  MoveL 6990 to (509.6, 509.6, 14.4) mm, rotated rx 0 ry 90 rz 0 deg; joints [-12.688, -27.581, 110.091, -16.755, -81.963, 51.382]
  Call Extruder(0.559)
  MoveL 6991 to (490.4, 509.6, 14.4) mm, rotated rx 0 ry 90 rz 0 deg; joints [-13.088, -27.943, 112.38, -17.087, -83.818, 50.861]
  MoveL 6992 to (490.4, 490.4, 14.4) mm, rotated rx 0 ry 90 rz 0 deg; joints [-11.303, -28.014, 112.87, -15.281, -84.175, 50.582]
  Call Extruder(0.146)
  MoveL 6993 to (495.43, 490.4, 14.4) mm, rotated rx 0 ry 90 rz 0 deg; joints [-11.21, -27.928, 112.274, -15.202, -83.681, 50.708]
  Call Extruder(0.010)
  MoveL 6994 to (495.78, 490.4, 14.4) mm, rotated rx 0 ry 90 rz 0 deg; joints [-11.203, -27.922, 112.232, -15.196, -83.646, 50.717]
  Call Extruder(0.007)
  MoveL 6995 to (495.78, 490.75, 14.4) mm, rotated rx 0 ry 90 rz 0 deg; joints [-11.236, -27.92, 112.224, -15.229, -83.64, 50.722]
  Call Extruder(0.035)
  MoveL 6996 to (495.78, 491.95, 14.4) mm, rotated rx 0 ry 90 rz 0 deg; joints [-11.347, -27.916, 112.196, -15.342, -83.62, 50.739]
  Call Extruder(0.010)
  MoveL 6997 to (495.78, 492.3, 14.4) mm, rotated rx 0 ry 90 rz 0 deg; joints [-11.38, -27.915, 112.187, -15.375, -83.614, 50.744]
  Call Extruder(0.007)
  MoveL 6998 to (496.13, 492.3, 14.4) mm, rotated rx 0 ry 90 rz 0 deg; joints [-11.373, -27.909, 112.146, -15.369, -83.58, 50.753]
  Call Extruder(0.061)
  MoveL 6999 to (498.23, 492.3, 14.4) mm, rotated rx 0 ry 90 rz 0 deg; joints [-11.334, -27.871, 111.895, -15.336, -83.373, 50.806]
  Call Extruder(0.055)
  MoveL 7000 to (498.23, 490.4, 14.4) mm, rotated rx 0 ry 90 rz 0 deg; joints [-11.158, -27.878, 111.94, -15.158, -83.405, 50.778]
  Call Extruder(0.082)
  MoveL 7001 to (501.04, 490.4, 14.4) mm, rotated rx 0 ry 90 rz 0 deg; joints [-11.107, -27.827, 111.605, -15.116, -83.13, 50.848]
  Call Extruder(0.055)
  MoveL 7002 to (501.04, 492.3, 14.4) mm, rotated rx 0 ry 90 rz 0 deg; joints [-11.282, -27.82, 111.56, -15.293, -83.098, 50.876]
  Call Extruder(0.061)
  MoveL 7003 to (503.12, 492.3, 14.4) mm, rotated rx 0 ry 90 rz 0 deg; joints [-11.244, -27.781, 111.31, -15.262, -82.893, 50.928]
  Call Extruder(0.007)
  MoveL 7004 to (503.48, 492.3, 14.4) mm, rotated rx 0 ry 90 rz 0 deg; joints [-11.238, -27.774, 111.268, -15.256, -82.859, 50.937]
  Set speed (120.0 mm/s)
  MoveL 7005 to (503.48, 491.95, 14.4) mm, rotated rx 0 ry 90 rz 0 deg; joints [-11.206, -27.775, 111.276, -15.224, -82.865, 50.931]
  Set speed (1000.0 mm/s)
  MoveL 7006 to (503.47, 491.9, 14.4) mm, rotated rx 0 ry 90 rz 0 deg; joints [-11.201, -27.775, 111.278, -15.219, -82.866, 50.931]
  Set speed (1000.0 mm/s)
  MoveL 7007 to (504.18, 491.9, 14.4) mm, rotated rx 0 ry 90 rz 0 deg; joints [-11.189, -27.762, 111.194, -15.209, -82.797, 50.948]
  Set speed (1000.0 mm/s)
  MoveL 7008 to (495.75, 492.33, 14.4) mm, rotated rx 0 ry 90 rz 0 deg; joints [-11.383, -27.915, 112.19, -15.378, -83.616, 50.744]
  Set speed (1000.0 mm/s)
  MoveL 7009 to (490.68, 490.68, 14.4) mm, rotated rx 0 ry 90 rz 0 deg; joints [-11.324, -28.008, 112.831, -15.303, -84.143, 50.593]
  Set speed (1000.0 mm/s)
  MoveL 7010 to (490.68, 490.68, 14.5) mm, rotated rx 0 ry 90 rz 0 deg; joints [-11.324, -28.019, 112.836, -15.303, -84.138, 50.594]
  Set speed (30.0 mm/s)
  Call Extruder(0.767)
  MoveL 7011 to (509.32, 509.32, 14.5) mm, rotated rx 0 ry 90 rz 0 deg; joints [-12.669, -27.598, 110.138, -16.734, -81.99, 51.371]
  MoveL 7012 to (509.44, 509.44, 14.5) mm, rotated rx 0 ry 90 rz 0 deg; joints [-12.677, -27.595, 110.12, -16.743, -81.976, 51.376]
  Set speed (120.0 mm/s)
  MoveL 7013 to (507.64, 503.83, 14.5) mm, rotated rx 0 ry 90 rz 0 deg; joints [-12.208, -27.657, 110.485, -16.258, -82.25, 51.231]
  Set speed (1000.0 mm/s)
  MoveL 7014 to (507.39, 502.51, 14.5) mm, rotated rx 0 ry 90 rz 0 deg; joints [-12.093, -27.667, 110.55, -16.14, -82.298, 51.202]
  Set speed (30.0 mm/s)
  Call Extruder(0.280)
  MoveL 7015 to (500.58, 509.32, 14.5) mm, rotated rx 0 ry 90 rz 0 deg; joints [-12.847, -27.771, 111.185, -16.88, -82.834, 51.137]
  Set speed (120.0 mm/s)
  MoveL 7016 to (499.42, 509.32, 14.5) mm, rotated rx 0 ry 90 rz 0 deg; joints [-12.872, -27.792, 111.324, -16.9, -82.946, 51.105]
  Set speed (30.0 mm/s)
  Call Extruder(0.360)
  MoveL 7017 to (490.68, 500.58, 14.5) mm, rotated rx 0 ry 90 rz 0 deg; joints [-12.247, -27.984, 112.592, -16.236, -83.959, 50.734]
  Set speed (120.0 mm/s)
  MoveL 7018 to (490.68, 499.42, 14.5) mm, rotated rx 0 ry 90 rz 0 deg; joints [-12.139, -27.988, 112.621, -16.127, -83.981, 50.717]
  Set speed (30.0 mm/s)
  Call Extruder(0.281)
  MoveL 7019 to (497.52, 492.58, 14.5) mm, rotated rx 0 ry 90 rz 0 deg; joints [-11.373, -27.894, 111.979, -15.374, -83.433, 50.794]
  Set speed (120.0 mm/s)
  MoveL 7020 to (498.45, 491.65, 14.5) mm, rotated rx 0 ry 90 rz 0 deg; joints [-11.269, -27.88, 111.889, -15.272, -83.357, 50.803]
  Set speed (30.0 mm/s)
  Call Extruder(0.040)
  MoveL 7021 to (499.42, 490.68, 14.5) mm, rotated rx 0 ry 90 rz 0 deg; joints [-11.163, -27.866, 111.797, -15.167, -83.279, 50.813]
  Set speed (120.0 mm/s)
  MoveL 7022 to (500.58, 490.68, 14.5) mm, rotated rx 0 ry 90 rz 0 deg; joints [-11.142, -27.845, 111.658, -15.149, -83.165, 50.842]
  Set speed (30.0 mm/s)
  Call Extruder(0.010)
  MoveL 7023 to (500.82, 490.92, 14.5) mm, rotated rx 0 ry 90 rz 0 deg; joints [-11.159, -27.839, 111.624, -15.168, -83.137, 50.852]
  Set speed (120.0 mm/s)
  MoveL 7024 to (501.08, 492.33, 14.5) mm, rotated rx 0 ry 90 rz 0 deg; joints [-11.284, -27.829, 111.56, -15.295, -83.089, 50.879]
  Set speed (1000.0 mm/s)
  MoveL 7025 to (502.48, 492.58, 14.5) mm, rotated rx 0 ry 90 rz 0 deg; joints [-11.282, -27.802, 111.386, -15.297, -82.947, 50.918]
  Set speed (30.0 mm/s)
  Call Extruder(0.202)
  MoveL 7026 to (507.39, 497.49, 14.5) mm, rotated rx 0 ry 90 rz 0 deg; joints [-11.639, -27.688, 110.677, -15.678, -82.384, 51.119]
  Set speed (120.0 mm/s)
  MoveL 7027 to (507.94, 498.04, 14.5) mm, rotated rx 0 ry 90 rz 0 deg; joints [-11.678, -27.675, 110.597, -15.72, -82.322, 51.141]
  Set speed (30.0 mm/s)
  Call Extruder(0.057)
  MoveL 7028 to (509.32, 499.42, 14.5) mm, rotated rx 0 ry 90 rz 0 deg; joints [-11.777, -27.642, 110.396, -15.826, -82.164, 51.199]
  Set speed (120.0 mm/s)
  MoveL 7029 to (509.32, 500.58, 14.5) mm, rotated rx 0 ry 90 rz 0 deg; joints [-11.882, -27.637, 110.367, -15.932, -82.144, 51.219]
  Set speed (30.0 mm/s)
  Call Extruder(0.018)
  MoveL 7030 to (508.87, 501.02, 14.5) mm, rotated rx 0 ry 90 rz 0 deg; joints [-11.931, -27.644, 110.409, -15.98, -82.18, 51.215]
  Set speed (120.0 mm/s)
  MoveL 7031 to (507.64, 497.79, 14.5) mm, rotated rx 0 ry 90 rz 0 deg; joints [-11.661, -27.682, 110.639, -15.701, -82.355, 51.13]
  Set speed (1000.0 mm/s)
  MoveL 7032 to (507.64, 495.21, 14.5) mm, rotated rx 0 ry 90 rz 0 deg; joints [-11.427, -27.692, 110.702, -15.464, -82.398, 51.088]
  Set speed (1000.0 mm/s)
  MoveL 7033 to (509.32, 490.68, 14.5) mm, rotated rx 0 ry 90 rz 0 deg; joints [-10.985, -27.677, 110.608, -15.021, -82.308, 51.056]
  Set speed (30.0 mm/s)
  Call Extruder(0.767)
  MoveL 7034 to (490.68, 509.32, 14.5) mm, rotated rx 0 ry 90 rz 0 deg; joints [-13.056, -27.95, 112.36, -17.056, -83.792, 50.865]
  MoveL 7035 to (490.56, 509.44, 14.5) mm, rotated rx 0 ry 90 rz 0 deg; joints [-13.07, -27.952, 112.371, -17.07, -83.801, 50.864]
  Set speed (120.0 mm/s)
  MoveL 7036 to (503.61, 492.37, 14.5) mm, rotated rx 0 ry 90 rz 0 deg; joints [-11.242, -27.782, 111.255, -15.261, -82.84, 50.943]
  Set speed (1000.0 mm/s)
  MoveL 7037 to (503.54, 492.3, 14.5) mm, rotated rx 0 ry 90 rz 0 deg; joints [-11.237, -27.783, 111.266, -15.255, -82.848, 50.94]
  Set speed (15.0 mm/s)
  Call Extruder(0.010)
  MoveL 7038 to (503.54, 491.95, 14.5) mm, rotated rx 0 ry 90 rz 0 deg; joints [-11.205, -27.785, 111.274, -15.223, -82.853, 50.934]
  Call Extruder(0.035)
  MoveL 7039 to (503.54, 490.75, 14.5) mm, rotated rx 0 ry 90 rz 0 deg; joints [-11.095, -27.789, 111.302, -15.111, -82.873, 50.916]
  Call Extruder(0.010)
  MoveL 7040 to (503.54, 490.4, 14.5) mm, rotated rx 0 ry 90 rz 0 deg; joints [-11.062, -27.79, 111.311, -15.079, -82.879, 50.911]
  Call Extruder(0.007)
  MoveL 7041 to (503.89, 490.4, 14.5) mm, rotated rx 0 ry 90 rz 0 deg; joints [-11.056, -27.784, 111.269, -15.074, -82.845, 50.919]
  Call Extruder(0.166)
  MoveL 7042 to (509.6, 490.4, 14.5) mm, rotated rx 0 ry 90 rz 0 deg; joints [-10.955, -27.672, 110.581, -14.991, -82.285, 51.058]
  Call Extruder(0.141)
  MoveL 7043 to (509.6, 495.24, 14.5) mm, rotated rx 0 ry 90 rz 0 deg; joints [-11.394, -27.653, 110.466, -15.437, -82.207, 51.137]
  Call Extruder(0.056)
  MoveL 7044 to (507.67, 495.24, 14.5) mm, rotated rx 0 ry 90 rz 0 deg; joints [-11.429, -27.692, 110.698, -15.466, -82.395, 51.089]
  Call Extruder(0.073)
  MoveL 7045 to (507.67, 497.76, 14.5) mm, rotated rx 0 ry 90 rz 0 deg; joints [-11.658, -27.682, 110.636, -15.698, -82.352, 51.13]
  Call Extruder(0.056)
  MoveL 7046 to (509.6, 497.76, 14.5) mm, rotated rx 0 ry 90 rz 0 deg; joints [-11.622, -27.643, 110.404, -15.669, -82.165, 51.179]
  Call Extruder(0.093)
  MoveL 7047 to (509.6, 500.95, 14.5) mm, rotated rx 0 ry 90 rz 0 deg; joints [-11.91, -27.63, 110.324, -15.963, -82.11, 51.232]
  Call Extruder(0.010)
  MoveL 7048 to (509.6, 501.3, 14.5) mm, rotated rx 0 ry 90 rz 0 deg; joints [-11.942, -27.628, 110.315, -15.995, -82.104, 51.238]
  Call Extruder(0.007)
  MoveL 7049 to (509.25, 501.3, 14.5) mm, rotated rx 0 ry 90 rz 0 deg; joints [-11.949, -27.635, 110.357, -16, -82.138, 51.229]
  Call Extruder(0.036)
  MoveL 7050 to (508.02, 501.3, 14.5) mm, rotated rx 0 ry 90 rz 0 deg; joints [-11.972, -27.66, 110.505, -16.019, -82.258, 51.198]
  Call Extruder(0.010)
  MoveL 7051 to (507.67, 501.3, 14.5) mm, rotated rx 0 ry 90 rz 0 deg; joints [-11.979, -27.667, 110.547, -16.024, -82.292, 51.189]
  Call Extruder(0.007)
  MoveL 7052 to (507.67, 501.65, 14.5) mm, rotated rx 0 ry 90 rz 0 deg; joints [-12.01, -27.665, 110.538, -16.057, -82.286, 51.195]
  Call Extruder(0.063)
  MoveL 7053 to (507.67, 503.81, 14.5) mm, rotated rx 0 ry 90 rz 0 deg; joints [-12.205, -27.656, 110.483, -16.255, -82.248, 51.231]
  Call Extruder(0.056)
  MoveL 7054 to (509.6, 503.81, 14.5) mm, rotated rx 0 ry 90 rz 0 deg; joints [-12.168, -27.617, 110.25, -16.225, -82.061, 51.281]
  Call Extruder(0.169)
  MoveL 7055 to (509.6, 509.6, 14.5) mm, rotated rx 0 ry 90 rz 0 deg; joints [-12.688, -27.591, 110.096, -16.755, -81.957, 51.383]
  Call Extruder(0.559)
  MoveL 7056 to (490.4, 509.6, 14.5) mm, rotated rx 0 ry 90 rz 0 deg; joints [-13.088, -27.954, 112.385, -17.088, -83.813, 50.862]
  MoveL 7057 to (490.4, 490.4, 14.5) mm, rotated rx 0 ry 90 rz 0 deg; joints [-11.303, -28.024, 112.875, -15.281, -84.17, 50.583]
  Call Extruder(0.145)
  MoveL 7058 to (495.37, 490.4, 14.5) mm, rotated rx 0 ry 90 rz 0 deg; joints [-11.211, -27.939, 112.286, -15.203, -83.681, 50.708]
  Call Extruder(0.010)
  MoveL 7059 to (495.72, 490.4, 14.5) mm, rotated rx 0 ry 90 rz 0 deg; joints [-11.204, -27.933, 112.244, -15.197, -83.646, 50.717]
  Call Extruder(0.007)
  MoveL 7060 to (495.72, 490.75, 14.5) mm, rotated rx 0 ry 90 rz 0 deg; joints [-11.237, -27.932, 112.236, -15.23, -83.641, 50.722]
  Call Extruder(0.035)
  MoveL 7061 to (495.72, 491.95, 14.5) mm, rotated rx 0 ry 90 rz 0 deg; joints [-11.348, -27.928, 112.208, -15.343, -83.62, 50.739]
  Call Extruder(0.010)
  MoveL 7062 to (495.72, 492.3, 14.5) mm, rotated rx 0 ry 90 rz 0 deg; joints [-11.381, -27.927, 112.199, -15.376, -83.614, 50.744]
  Call Extruder(0.007)
  MoveL 7063 to (496.07, 492.3, 14.5) mm, rotated rx 0 ry 90 rz 0 deg; joints [-11.374, -27.92, 112.158, -15.37, -83.58, 50.753]
  Call Extruder(0.061)
  MoveL 7064 to (498.17, 492.3, 14.5) mm, rotated rx 0 ry 90 rz 0 deg; joints [-11.335, -27.883, 111.907, -15.337, -83.373, 50.806]
  Call Extruder(0.055)
  MoveL 7065 to (498.18, 490.4, 14.5) mm, rotated rx 0 ry 90 rz 0 deg; joints [-11.159, -27.889, 111.952, -15.159, -83.405, 50.778]
  Call Extruder(0.085)
  MoveL 7066 to (501.1, 490.4, 14.5) mm, rotated rx 0 ry 90 rz 0 deg; joints [-11.106, -27.836, 111.602, -15.115, -83.118, 50.851]
  Call Extruder(0.055)
  MoveL 7067 to (501.1, 492.3, 14.5) mm, rotated rx 0 ry 90 rz 0 deg; joints [-11.281, -27.829, 111.557, -15.292, -83.086, 50.879]
  Call Extruder(0.061)
  MoveL 7068 to (503.19, 492.3, 14.5) mm, rotated rx 0 ry 90 rz 0 deg; joints [-11.243, -27.79, 111.307, -15.261, -82.882, 50.931]
  Call Extruder(0.007)
  MoveL 7069 to (503.54, 492.3, 14.5) mm, rotated rx 0 ry 90 rz 0 deg; joints [-11.237, -27.783, 111.266, -15.255, -82.848, 50.94]
  Set speed (120.0 mm/s)
  MoveL 7070 to (503.54, 491.95, 14.5) mm, rotated rx 0 ry 90 rz 0 deg; joints [-11.205, -27.785, 111.274, -15.223, -82.853, 50.934]
  Set speed (1000.0 mm/s)
  MoveL 7071 to (503.54, 491.9, 14.5) mm, rotated rx 0 ry 90 rz 0 deg; joints [-11.2, -27.785, 111.275, -15.218, -82.854, 50.934]
  Set speed (1000.0 mm/s)
  MoveL 7072 to (504.24, 491.9, 14.5) mm, rotated rx 0 ry 90 rz 0 deg; joints [-11.187, -27.771, 111.191, -15.208, -82.786, 50.951]
  Set speed (1000.0 mm/s)
  MoveL 7073 to (495.69, 492.33, 14.5) mm, rotated rx 0 ry 90 rz 0 deg; joints [-11.384, -27.927, 112.202, -15.379, -83.616, 50.744]
  Set speed (1000.0 mm/s)
  MoveL 7074 to (490.68, 490.68, 14.5) mm, rotated rx 0 ry 90 rz 0 deg; joints [-11.324, -28.019, 112.836, -15.303, -84.138, 50.594]
  Set speed (1000.0 mm/s)
  MoveL 7075 to (490.68, 490.68, 14.6) mm, rotated rx 0 ry 90 rz 0 deg; joints [-11.324, -28.029, 112.841, -15.303, -84.132, 50.596]
  Set speed (30.0 mm/s)
  Call Extruder(0.767)
  MoveL 7076 to (509.32, 509.32, 14.6) mm, rotated rx 0 ry 90 rz 0 deg; joints [-12.669, -27.609, 110.143, -16.734, -81.985, 51.372]
  MoveL 7077 to (509.44, 509.44, 14.6) mm, rotated rx 0 ry 90 rz 0 deg; joints [-12.677, -27.605, 110.125, -16.743, -81.97, 51.378]
  Set speed (120.0 mm/s)
  MoveL 7078 to (507.64, 503.89, 14.6) mm, rotated rx 0 ry 90 rz 0 deg; joints [-12.213, -27.667, 110.489, -16.263, -82.244, 51.234]
  Set speed (1000.0 mm/s)
  MoveL 7079 to (507.39, 502.51, 14.6) mm, rotated rx 0 ry 90 rz 0 deg; joints [-12.093, -27.678, 110.555, -16.14, -82.293, 51.204]
  Set speed (30.0 mm/s)
  Call Extruder(0.280)
  MoveL 7080 to (500.58, 509.32, 14.6) mm, rotated rx 0 ry 90 rz 0 deg; joints [-12.847, -27.781, 111.191, -16.88, -82.829, 51.138]
  Set speed (120.0 mm/s)
  MoveL 7081 to (499.42, 509.32, 14.6) mm, rotated rx 0 ry 90 rz 0 deg; joints [-12.872, -27.803, 111.329, -16.901, -82.941, 51.107]
  Set speed (30.0 mm/s)
  Call Extruder(0.360)
  MoveL 7082 to (490.68, 500.58, 14.6) mm, rotated rx 0 ry 90 rz 0 deg; joints [-12.247, -27.995, 112.597, -16.237, -83.954, 50.735]
  Set speed (120.0 mm/s)
  MoveL 7083 to (490.68, 499.42, 14.6) mm, rotated rx 0 ry 90 rz 0 deg; joints [-12.139, -27.999, 112.626, -16.128, -83.975, 50.718]
  Set speed (30.0 mm/s)
  Call Extruder(0.281)
  MoveL 7084 to (497.52, 492.58, 14.6) mm, rotated rx 0 ry 90 rz 0 deg; joints [-11.373, -27.904, 111.984, -15.374, -83.428, 50.795]
  Set speed (120.0 mm/s)
  MoveL 7085 to (498.4, 491.7, 14.6) mm, rotated rx 0 ry 90 rz 0 deg; joints [-11.276, -27.891, 111.9, -15.278, -83.356, 50.804]
  Set speed (30.0 mm/s)
  Call Extruder(0.042)
  MoveL 7086 to (499.42, 490.68, 14.6) mm, rotated rx 0 ry 90 rz 0 deg; joints [-11.163, -27.877, 111.802, -15.167, -83.273, 50.815]
  Set speed (120.0 mm/s)
  MoveL 7087 to (500.58, 490.68, 14.6) mm, rotated rx 0 ry 90 rz 0 deg; joints [-11.141, -27.855, 111.663, -15.149, -83.159, 50.843]
  Set speed (30.0 mm/s)
  Call Extruder(0.013)
  MoveL 7088 to (500.89, 490.99, 14.6) mm, rotated rx 0 ry 90 rz 0 deg; joints [-11.164, -27.848, 111.62, -15.173, -83.124, 50.855]
  Set speed (120.0 mm/s)
  MoveL 7089 to (502.48, 492.58, 14.6) mm, rotated rx 0 ry 90 rz 0 deg; joints [-11.282, -27.813, 111.391, -15.298, -82.941, 50.919]
  Set speed (30.0 mm/s)
  Call Extruder(0.202)
  MoveL 7090 to (507.39, 497.49, 14.6) mm, rotated rx 0 ry 90 rz 0 deg; joints [-11.639, -27.699, 110.681, -15.678, -82.379, 51.12]
  Set speed (120.0 mm/s)
  MoveL 7091 to (507.88, 497.98, 14.6) mm, rotated rx 0 ry 90 rz 0 deg; joints [-11.674, -27.687, 110.611, -15.716, -82.323, 51.14]
  Set speed (30.0 mm/s)
  Call Extruder(0.059)
  MoveL 7092 to (509.32, 499.42, 14.6) mm, rotated rx 0 ry 90 rz 0 deg; joints [-11.777, -27.652, 110.401, -15.826, -82.159, 51.201]
  Set speed (120.0 mm/s)
  MoveL 7093 to (509.32, 500.58, 14.6) mm, rotated rx 0 ry 90 rz 0 deg; joints [-11.882, -27.647, 110.372, -15.933, -82.139, 51.22]
  Set speed (30.0 mm/s)
  Call Extruder(0.021)
  MoveL 7094 to (508.82, 501.08, 14.6) mm, rotated rx 0 ry 90 rz 0 deg; joints [-11.937, -27.655, 110.42, -15.986, -82.179, 51.216]
  Set speed (120.0 mm/s)
  MoveL 7095 to (507.65, 497.73, 14.6) mm, rotated rx 0 ry 90 rz 0 deg; joints [-11.656, -27.693, 110.645, -15.696, -82.35, 51.13]
  Set speed (1000.0 mm/s)
  MoveL 7096 to (507.64, 495.15, 14.6) mm, rotated rx 0 ry 90 rz 0 deg; joints [-11.422, -27.703, 110.709, -15.458, -82.394, 51.088]
  Set speed (1000.0 mm/s)
  MoveL 7097 to (509.32, 490.68, 14.6) mm, rotated rx 0 ry 90 rz 0 deg; joints [-10.985, -27.687, 110.614, -15.021, -82.303, 51.057]
  Set speed (30.0 mm/s)
  Call Extruder(0.767)
  MoveL 7098 to (490.68, 509.32, 14.6) mm, rotated rx 0 ry 90 rz 0 deg; joints [-13.056, -27.961, 112.365, -17.056, -83.786, 50.867]
  MoveL 7099 to (490.56, 509.44, 14.6) mm, rotated rx 0 ry 90 rz 0 deg; joints [-13.07, -27.962, 112.376, -17.07, -83.796, 50.866]
  Set speed (120.0 mm/s)
  MoveL 7100 to (503.67, 492.37, 14.6) mm, rotated rx 0 ry 90 rz 0 deg; joints [-11.241, -27.791, 111.253, -15.26, -82.828, 50.946]
  Set speed (1000.0 mm/s)
  MoveL 7101 to (503.6, 492.3, 14.6) mm, rotated rx 0 ry 90 rz 0 deg; joints [-11.236, -27.793, 111.263, -15.255, -82.836, 50.943]
  Set speed (15.0 mm/s)
  Call Extruder(0.010)
  MoveL 7102 to (503.6, 491.95, 14.6) mm, rotated rx 0 ry 90 rz 0 deg; joints [-11.203, -27.794, 111.271, -15.222, -82.842, 50.937]
  Call Extruder(0.035)
  MoveL 7103 to (503.6, 490.75, 14.6) mm, rotated rx 0 ry 90 rz 0 deg; joints [-11.093, -27.798, 111.3, -15.111, -82.862, 50.919]
  Call Extruder(0.010)
  MoveL 7104 to (503.6, 490.4, 14.6) mm, rotated rx 0 ry 90 rz 0 deg; joints [-11.061, -27.8, 111.308, -15.078, -82.868, 50.914]
  Call Extruder(0.007)
  MoveL 7105 to (503.95, 490.4, 14.6) mm, rotated rx 0 ry 90 rz 0 deg; joints [-11.055, -27.793, 111.266, -15.073, -82.833, 50.922]
  Call Extruder(0.164)
  MoveL 7106 to (509.6, 490.4, 14.6) mm, rotated rx 0 ry 90 rz 0 deg; joints [-10.955, -27.683, 110.586, -14.991, -82.28, 51.06]
  Call Extruder(0.139)
  MoveL 7107 to (509.6, 495.18, 14.6) mm, rotated rx 0 ry 90 rz 0 deg; joints [-11.388, -27.664, 110.472, -15.432, -82.203, 51.137]
  Call Extruder(0.056)
  MoveL 7108 to (507.67, 495.18, 14.6) mm, rotated rx 0 ry 90 rz 0 deg; joints [-11.424, -27.702, 110.705, -15.46, -82.391, 51.089]
  Call Extruder(0.073)
  MoveL 7109 to (507.67, 497.7, 14.6) mm, rotated rx 0 ry 90 rz 0 deg; joints [-11.652, -27.692, 110.642, -15.693, -82.348, 51.131]
  Call Extruder(0.046)
  MoveL 7110 to (509.25, 497.7, 14.6) mm, rotated rx 0 ry 90 rz 0 deg; joints [-11.623, -27.661, 110.453, -15.669, -82.195, 51.17]
  Call Extruder(0.010)
  MoveL 7111 to (509.6, 497.7, 14.6) mm, rotated rx 0 ry 90 rz 0 deg; joints [-11.616, -27.654, 110.41, -15.664, -82.161, 51.179]
  Call Extruder(0.007)
  MoveL 7112 to (509.6, 498.05, 14.6) mm, rotated rx 0 ry 90 rz 0 deg; joints [-11.648, -27.652, 110.402, -15.696, -82.155, 51.185]
  Call Extruder(0.086)
  MoveL 7113 to (509.6, 501.01, 14.6) mm, rotated rx 0 ry 90 rz 0 deg; joints [-11.915, -27.64, 110.327, -15.968, -82.104, 51.235]
  Call Extruder(0.010)
  MoveL 7114 to (509.6, 501.36, 14.6) mm, rotated rx 0 ry 90 rz 0 deg; joints [-11.947, -27.638, 110.318, -16, -82.098, 51.241]
  Call Extruder(0.007)
  MoveL 7115 to (509.25, 501.36, 14.6) mm, rotated rx 0 ry 90 rz 0 deg; joints [-11.954, -27.645, 110.361, -16.006, -82.132, 51.232]
  Call Extruder(0.036)
  MoveL 7116 to (508.02, 501.36, 14.6) mm, rotated rx 0 ry 90 rz 0 deg; joints [-11.977, -27.67, 110.509, -16.024, -82.252, 51.2]
  Call Extruder(0.010)
  MoveL 7117 to (507.67, 501.36, 14.6) mm, rotated rx 0 ry 90 rz 0 deg; joints [-11.984, -27.677, 110.551, -16.03, -82.286, 51.191]
  Call Extruder(0.007)
  MoveL 7118 to (507.67, 501.71, 14.6) mm, rotated rx 0 ry 90 rz 0 deg; joints [-12.015, -27.676, 110.542, -16.062, -82.28, 51.197]
  Call Extruder(0.063)
  MoveL 7119 to (507.67, 503.86, 14.6) mm, rotated rx 0 ry 90 rz 0 deg; joints [-12.21, -27.666, 110.486, -16.26, -82.242, 51.234]
  Call Extruder(0.056)
  MoveL 7120 to (509.6, 503.87, 14.6) mm, rotated rx 0 ry 90 rz 0 deg; joints [-12.173, -27.627, 110.254, -16.23, -82.055, 51.284]
  Call Extruder(0.167)
  MoveL 7121 to (509.6, 509.6, 14.6) mm, rotated rx 0 ry 90 rz 0 deg; joints [-12.688, -27.602, 110.101, -16.755, -81.952, 51.385]
  Call Extruder(0.559)
  MoveL 7122 to (490.4, 509.6, 14.6) mm, rotated rx 0 ry 90 rz 0 deg; joints [-13.088, -27.965, 112.39, -17.088, -83.808, 50.864]
  MoveL 7123 to (490.4, 490.4, 14.6) mm, rotated rx 0 ry 90 rz 0 deg; joints [-11.303, -28.035, 112.881, -15.281, -84.165, 50.585]
  Call Extruder(0.143)
  MoveL 7124 to (495.31, 490.4, 14.6) mm, rotated rx 0 ry 90 rz 0 deg; joints [-11.212, -27.951, 112.298, -15.204, -83.681, 50.708]
  Call Extruder(0.010)
  MoveL 7125 to (495.66, 490.4, 14.6) mm, rotated rx 0 ry 90 rz 0 deg; joints [-11.205, -27.945, 112.256, -15.198, -83.647, 50.717]
  Call Extruder(0.007)
  MoveL 7126 to (495.66, 490.75, 14.6) mm, rotated rx 0 ry 90 rz 0 deg; joints [-11.238, -27.944, 112.248, -15.231, -83.641, 50.722]
  Call Extruder(0.035)
  MoveL 7127 to (495.66, 491.95, 14.6) mm, rotated rx 0 ry 90 rz 0 deg; joints [-11.349, -27.939, 112.22, -15.344, -83.621, 50.739]
  Call Extruder(0.010)
  MoveL 7128 to (495.66, 492.3, 14.6) mm, rotated rx 0 ry 90 rz 0 deg; joints [-11.382, -27.938, 112.211, -15.377, -83.615, 50.744]
  Call Extruder(0.007)
  MoveL 7129 to (496.01, 492.3, 14.6) mm, rotated rx 0 ry 90 rz 0 deg; joints [-11.375, -27.932, 112.17, -15.371, -83.58, 50.753]
  Call Extruder(0.061)
  MoveL 7130 to (498.12, 492.3, 14.6) mm, rotated rx 0 ry 90 rz 0 deg; joints [-11.336, -27.894, 111.919, -15.339, -83.374, 50.806]
  Call Extruder(0.055)
  MoveL 7131 to (498.12, 490.4, 14.6) mm, rotated rx 0 ry 90 rz 0 deg; joints [-11.16, -27.901, 111.964, -15.16, -83.406, 50.778]
  Call Extruder(0.089)
  MoveL 7132 to (501.16, 490.4, 14.6) mm, rotated rx 0 ry 90 rz 0 deg; joints [-11.105, -27.845, 111.6, -15.114, -83.107, 50.854]
  Call Extruder(0.055)
  MoveL 7133 to (501.17, 492.3, 14.6) mm, rotated rx 0 ry 90 rz 0 deg; joints [-11.28, -27.838, 111.555, -15.292, -83.075, 50.882]
  Call Extruder(0.061)
  MoveL 7134 to (503.25, 492.3, 14.6) mm, rotated rx 0 ry 90 rz 0 deg; joints [-11.242, -27.799, 111.305, -15.26, -82.87, 50.934]
  Call Extruder(0.007)
  MoveL 7135 to (503.6, 492.3, 14.6) mm, rotated rx 0 ry 90 rz 0 deg; joints [-11.236, -27.793, 111.263, -15.255, -82.836, 50.943]
  Set speed (120.0 mm/s)
  MoveL 7136 to (503.6, 491.95, 14.6) mm, rotated rx 0 ry 90 rz 0 deg; joints [-11.203, -27.794, 111.271, -15.222, -82.842, 50.937]
  Set speed (1000.0 mm/s)
  MoveL 7137 to (503.6, 491.9, 14.6) mm, rotated rx 0 ry 90 rz 0 deg; joints [-11.199, -27.794, 111.272, -15.218, -82.843, 50.937]
  Set speed (1000.0 mm/s)
  MoveL 7138 to (504.3, 491.9, 14.6) mm, rotated rx 0 ry 90 rz 0 deg; joints [-11.186, -27.781, 111.188, -15.207, -82.774, 50.954]
  Set speed (1000.0 mm/s)
  MoveL 7139 to (495.63, 492.33, 14.6) mm, rotated rx 0 ry 90 rz 0 deg; joints [-11.385, -27.939, 112.214, -15.38, -83.617, 50.744]
  Set speed (1000.0 mm/s)
  MoveL 7140 to (490.68, 490.68, 14.6) mm, rotated rx 0 ry 90 rz 0 deg; joints [-11.324, -28.029, 112.841, -15.303, -84.132, 50.596]
  Set speed (1000.0 mm/s)
  MoveL 7141 to (490.68, 490.68, 14.7) mm, rotated rx 0 ry 90 rz 0 deg; joints [-11.324, -28.04, 112.846, -15.303, -84.127, 50.597]
  Set speed (30.0 mm/s)
  Call Extruder(0.767)
  MoveL 7142 to (509.32, 509.32, 14.7) mm, rotated rx 0 ry 90 rz 0 deg; joints [-12.669, -27.619, 110.148, -16.734, -81.979, 51.374]
  MoveL 7143 to (509.44, 509.44, 14.7) mm, rotated rx 0 ry 90 rz 0 deg; joints [-12.677, -27.616, 110.13, -16.743, -81.965, 51.379]
  Set speed (120.0 mm/s)
  MoveL 7144 to (507.64, 503.95, 14.7) mm, rotated rx 0 ry 90 rz 0 deg; joints [-12.218, -27.677, 110.493, -16.269, -82.238, 51.236]
  Set speed (1000.0 mm/s)
  MoveL 7145 to (507.39, 502.51, 14.7) mm, rotated rx 0 ry 90 rz 0 deg; joints [-12.093, -27.688, 110.56, -16.14, -82.288, 51.205]
  Set speed (30.0 mm/s)
  Call Extruder(0.280)
  MoveL 7146 to (500.58, 509.32, 14.7) mm, rotated rx 0 ry 90 rz 0 deg; joints [-12.847, -27.792, 111.196, -16.881, -82.823, 51.14]
  Set speed (120.0 mm/s)
  MoveL 7147 to (499.42, 509.32, 14.7) mm, rotated rx 0 ry 90 rz 0 deg; joints [-12.872, -27.814, 111.334, -16.901, -82.935, 51.108]
  Set speed (30.0 mm/s)
  Call Extruder(0.360)
  MoveL 7148 to (490.68, 500.58, 14.7) mm, rotated rx 0 ry 90 rz 0 deg; joints [-12.247, -28.005, 112.602, -16.237, -83.949, 50.737]
  Set speed (120.0 mm/s)
  MoveL 7149 to (490.68, 499.42, 14.7) mm, rotated rx 0 ry 90 rz 0 deg; joints [-12.139, -28.009, 112.631, -16.128, -83.97, 50.72]
  Set speed (30.0 mm/s)
  Call Extruder(0.281)
  MoveL 7150 to (497.52, 492.58, 14.7) mm, rotated rx 0 ry 90 rz 0 deg; joints [-11.373, -27.915, 111.989, -15.374, -83.423, 50.797]
  Set speed (120.0 mm/s)
  MoveL 7151 to (498.34, 491.76, 14.7) mm, rotated rx 0 ry 90 rz 0 deg; joints [-11.282, -27.903, 111.91, -15.284, -83.356, 50.805]
  Set speed (30.0 mm/s)
  Call Extruder(0.044)
  MoveL 7152 to (499.42, 490.68, 14.7) mm, rotated rx 0 ry 90 rz 0 deg; joints [-11.163, -27.887, 111.807, -15.167, -83.268, 50.816]
  Set speed (120.0 mm/s)
  MoveL 7153 to (500.58, 490.68, 14.7) mm, rotated rx 0 ry 90 rz 0 deg; joints [-11.142, -27.866, 111.669, -15.149, -83.154, 50.845]
  Set speed (30.0 mm/s)
  Call Extruder(0.015)
  MoveL 7154 to (500.95, 491.05, 14.7) mm, rotated rx 0 ry 90 rz 0 deg; joints [-11.169, -27.858, 111.616, -15.178, -83.112, 50.859]
  Set speed (120.0 mm/s)
  MoveL 7155 to (502.48, 492.58, 14.7) mm, rotated rx 0 ry 90 rz 0 deg; joints [-11.282, -27.823, 111.396, -15.298, -82.936, 50.921]
  Set speed (30.0 mm/s)
  Call Extruder(0.202)
  MoveL 7156 to (507.39, 497.49, 14.7) mm, rotated rx 0 ry 90 rz 0 deg; joints [-11.639, -27.709, 110.687, -15.678, -82.374, 51.122]
  Set speed (120.0 mm/s)
  MoveL 7157 to (507.82, 497.92, 14.7) mm, rotated rx 0 ry 90 rz 0 deg; joints [-11.67, -27.699, 110.624, -15.711, -82.325, 51.139]
  Set speed (30.0 mm/s)
  Call Extruder(0.062)
  MoveL 7158 to (509.32, 499.42, 14.7) mm, rotated rx 0 ry 90 rz 0 deg; joints [-11.777, -27.663, 110.406, -15.826, -82.154, 51.202]
  Set speed (120.0 mm/s)
  MoveL 7159 to (509.32, 500.58, 14.7) mm, rotated rx 0 ry 90 rz 0 deg; joints [-11.882, -27.658, 110.377, -15.933, -82.134, 51.222]
  Set speed (30.0 mm/s)
  Call Extruder(0.023)
  MoveL 7160 to (508.76, 501.13, 14.7) mm, rotated rx 0 ry 90 rz 0 deg; joints [-11.943, -27.667, 110.43, -15.993, -82.178, 51.217]
  Set speed (120.0 mm/s)
  MoveL 7161 to (507.65, 497.67, 14.7) mm, rotated rx 0 ry 90 rz 0 deg; joints [-11.65, -27.703, 110.652, -15.691, -82.346, 51.131]
  Set speed (1000.0 mm/s)
  MoveL 7162 to (507.64, 495.09, 14.7) mm, rotated rx 0 ry 90 rz 0 deg; joints [-11.416, -27.714, 110.715, -15.453, -82.39, 51.089]
  Set speed (1000.0 mm/s)
  MoveL 7163 to (509.32, 490.68, 14.7) mm, rotated rx 0 ry 90 rz 0 deg; joints [-10.985, -27.698, 110.619, -15.021, -82.298, 51.059]
  Set speed (30.0 mm/s)
  Call Extruder(0.767)
  MoveL 7164 to (490.68, 509.32, 14.7) mm, rotated rx 0 ry 90 rz 0 deg; joints [-13.056, -27.972, 112.37, -17.056, -83.781, 50.869]
  MoveL 7165 to (490.56, 509.44, 14.7) mm, rotated rx 0 ry 90 rz 0 deg; joints [-13.07, -27.973, 112.381, -17.07, -83.791, 50.867]
  Set speed (120.0 mm/s)
  MoveL 7166 to (503.74, 492.37, 14.7) mm, rotated rx 0 ry 90 rz 0 deg; joints [-11.239, -27.8, 111.25, -15.259, -82.817, 50.949]
  Set speed (1000.0 mm/s)
  MoveL 7167 to (503.67, 492.3, 14.7) mm, rotated rx 0 ry 90 rz 0 deg; joints [-11.234, -27.802, 111.26, -15.254, -82.825, 50.946]
  Set speed (15.0 mm/s)
  Call Extruder(0.010)
  MoveL 7168 to (503.67, 491.95, 14.7) mm, rotated rx 0 ry 90 rz 0 deg; joints [-11.202, -27.803, 111.269, -15.221, -82.83, 50.94]
  Call Extruder(0.035)
  MoveL 7169 to (503.67, 490.75, 14.7) mm, rotated rx 0 ry 90 rz 0 deg; joints [-11.092, -27.808, 111.297, -15.11, -82.85, 50.922]
  Call Extruder(0.010)
  MoveL 7170 to (503.66, 490.4, 14.7) mm, rotated rx 0 ry 90 rz 0 deg; joints [-11.06, -27.809, 111.306, -15.077, -82.856, 50.917]
  Call Extruder(0.007)
  MoveL 7171 to (504.02, 490.4, 14.7) mm, rotated rx 0 ry 90 rz 0 deg; joints [-11.054, -27.802, 111.264, -15.072, -82.822, 50.925]
  Call Extruder(0.163)
  MoveL 7172 to (509.6, 490.4, 14.7) mm, rotated rx 0 ry 90 rz 0 deg; joints [-10.955, -27.693, 110.591, -14.991, -82.275, 51.061]
  Call Extruder(0.137)
  MoveL 7173 to (509.6, 495.12, 14.7) mm, rotated rx 0 ry 90 rz 0 deg; joints [-11.383, -27.675, 110.479, -15.426, -82.198, 51.138]
  Call Extruder(0.056)
  MoveL 7174 to (507.67, 495.12, 14.7) mm, rotated rx 0 ry 90 rz 0 deg; joints [-11.418, -27.713, 110.711, -15.455, -82.386, 51.09]
  Call Extruder(0.073)
  MoveL 7175 to (507.67, 497.64, 14.7) mm, rotated rx 0 ry 90 rz 0 deg; joints [-11.647, -27.703, 110.649, -15.688, -82.344, 51.131]
  Call Extruder(0.056)
  MoveL 7176 to (509.6, 497.64, 14.7) mm, rotated rx 0 ry 90 rz 0 deg; joints [-11.611, -27.664, 110.417, -15.659, -82.156, 51.18]
  Call Extruder(0.100)
  MoveL 7177 to (509.6, 501.07, 14.7) mm, rotated rx 0 ry 90 rz 0 deg; joints [-11.921, -27.65, 110.331, -15.973, -82.098, 51.237]
  Call Extruder(0.010)
  MoveL 7178 to (509.6, 501.42, 14.7) mm, rotated rx 0 ry 90 rz 0 deg; joints [-11.952, -27.648, 110.322, -16.006, -82.092, 51.243]
  Call Extruder(0.007)
  MoveL 7179 to (509.25, 501.42, 14.7) mm, rotated rx 0 ry 90 rz 0 deg; joints [-11.959, -27.656, 110.364, -16.011, -82.126, 51.234]
  Call Extruder(0.036)
  MoveL 7180 to (508.02, 501.41, 14.7) mm, rotated rx 0 ry 90 rz 0 deg; joints [-11.982, -27.68, 110.512, -16.03, -82.246, 51.203]
  Call Extruder(0.010)
  MoveL 7181 to (507.67, 501.41, 14.7) mm, rotated rx 0 ry 90 rz 0 deg; joints [-11.989, -27.687, 110.555, -16.035, -82.28, 51.194]
  Call Extruder(0.007)
  MoveL 7182 to (507.67, 501.76, 14.7) mm, rotated rx 0 ry 90 rz 0 deg; joints [-12.02, -27.686, 110.546, -16.067, -82.273, 51.2]
  Call Extruder(0.063)
  MoveL 7183 to (507.67, 503.92, 14.7) mm, rotated rx 0 ry 90 rz 0 deg; joints [-12.215, -27.677, 110.49, -16.266, -82.236, 51.236]
  Call Extruder(0.056)
  MoveL 7184 to (509.6, 503.92, 14.7) mm, rotated rx 0 ry 90 rz 0 deg; joints [-12.178, -27.638, 110.258, -16.235, -82.049, 51.286]
  Call Extruder(0.000)
  MoveL 7185 to (509.6, 503.92, 14.7) mm, rotated rx 0 ry 90 rz 0 deg; joints [-12.178, -27.638, 110.257, -16.235, -82.049, 51.286]
  Call Extruder(0.165)
  MoveL 7186 to (509.6, 509.6, 14.7) mm, rotated rx 0 ry 90 rz 0 deg; joints [-12.688, -27.612, 110.107, -16.755, -81.947, 51.386]
  Call Extruder(0.559)
  MoveL 7187 to (490.4, 509.6, 14.7) mm, rotated rx 0 ry 90 rz 0 deg; joints [-13.088, -27.975, 112.395, -17.088, -83.803, 50.865]
  MoveL 7188 to (490.4, 490.4, 14.7) mm, rotated rx 0 ry 90 rz 0 deg; joints [-11.303, -28.046, 112.886, -15.282, -84.159, 50.586]
  Call Extruder(0.141)
  MoveL 7189 to (495.26, 490.4, 14.7) mm, rotated rx 0 ry 90 rz 0 deg; joints [-11.213, -27.963, 112.31, -15.205, -83.681, 50.709]
  Call Extruder(0.010)
  MoveL 7190 to (495.61, 490.4, 14.7) mm, rotated rx 0 ry 90 rz 0 deg; joints [-11.206, -27.956, 112.268, -15.199, -83.647, 50.717]
  Call Extruder(0.007)
  MoveL 7191 to (495.61, 490.75, 14.7) mm, rotated rx 0 ry 90 rz 0 deg; joints [-11.239, -27.955, 112.26, -15.232, -83.641, 50.722]
  Call Extruder(0.035)
  MoveL 7192 to (495.61, 491.95, 14.7) mm, rotated rx 0 ry 90 rz 0 deg; joints [-11.35, -27.951, 112.231, -15.345, -83.621, 50.739]
  Call Extruder(0.010)
  MoveL 7193 to (495.61, 492.3, 14.7) mm, rotated rx 0 ry 90 rz 0 deg; joints [-11.383, -27.95, 112.223, -15.378, -83.615, 50.744]
  Call Extruder(0.007)
  MoveL 7194 to (495.96, 492.3, 14.7) mm, rotated rx 0 ry 90 rz 0 deg; joints [-11.376, -27.944, 112.181, -15.372, -83.58, 50.753]
  Call Extruder(0.061)
  MoveL 7195 to (498.06, 492.3, 14.7) mm, rotated rx 0 ry 90 rz 0 deg; joints [-11.337, -27.906, 111.931, -15.34, -83.374, 50.806]
  Call Extruder(0.055)
  MoveL 7196 to (498.06, 490.4, 14.7) mm, rotated rx 0 ry 90 rz 0 deg; joints [-11.162, -27.913, 111.976, -15.161, -83.406, 50.778]
  Call Extruder(0.092)
  MoveL 7197 to (501.23, 490.4, 14.7) mm, rotated rx 0 ry 90 rz 0 deg; joints [-11.104, -27.855, 111.598, -15.114, -83.095, 50.857]
  Call Extruder(0.055)
  MoveL 7198 to (501.23, 492.3, 14.7) mm, rotated rx 0 ry 90 rz 0 deg; joints [-11.279, -27.848, 111.552, -15.291, -83.063, 50.885]
  Call Extruder(0.061)
  MoveL 7199 to (503.32, 492.3, 14.7) mm, rotated rx 0 ry 90 rz 0 deg; joints [-11.241, -27.809, 111.302, -15.259, -82.859, 50.937]
  Call Extruder(0.007)
  MoveL 7200 to (503.67, 492.3, 14.7) mm, rotated rx 0 ry 90 rz 0 deg; joints [-11.234, -27.802, 111.26, -15.254, -82.825, 50.946]
  Set speed (120.0 mm/s)
  MoveL 7201 to (503.67, 491.95, 14.7) mm, rotated rx 0 ry 90 rz 0 deg; joints [-11.202, -27.803, 111.269, -15.221, -82.83, 50.94]
  Set speed (1000.0 mm/s)
  MoveL 7202 to (503.67, 491.9, 14.7) mm, rotated rx 0 ry 90 rz 0 deg; joints [-11.198, -27.803, 111.27, -15.217, -82.831, 50.94]
  Set speed (1000.0 mm/s)
  MoveL 7203 to (504.37, 491.9, 14.7) mm, rotated rx 0 ry 90 rz 0 deg; joints [-11.185, -27.79, 111.186, -15.206, -82.763, 50.957]
  Set speed (1000.0 mm/s)
  MoveL 7204 to (495.58, 492.33, 14.7) mm, rotated rx 0 ry 90 rz 0 deg; joints [-11.386, -27.95, 112.226, -15.381, -83.617, 50.744]
  Set speed (1000.0 mm/s)
  MoveL 7205 to (490.68, 490.68, 14.7) mm, rotated rx 0 ry 90 rz 0 deg; joints [-11.324, -28.04, 112.846, -15.303, -84.127, 50.597]
  Set speed (1000.0 mm/s)
  MoveL 7206 to (490.68, 490.68, 14.8) mm, rotated rx 0 ry 90 rz 0 deg; joints [-11.324, -28.051, 112.851, -15.304, -84.122, 50.599]
  Set speed (30.0 mm/s)
  Call Extruder(0.767)
  MoveL 7207 to (509.32, 509.32, 14.8) mm, rotated rx 0 ry 90 rz 0 deg; joints [-12.669, -27.629, 110.153, -16.734, -81.974, 51.375]
  MoveL 7208 to (509.44, 509.44, 14.8) mm, rotated rx 0 ry 90 rz 0 deg; joints [-12.677, -27.626, 110.135, -16.744, -81.96, 51.381]
  Set speed (120.0 mm/s)
  MoveL 7209 to (507.64, 504, 14.8) mm, rotated rx 0 ry 90 rz 0 deg; joints [-12.223, -27.687, 110.496, -16.274, -82.232, 51.238]
  Set speed (1000.0 mm/s)
  MoveL 7210 to (507.39, 502.51, 14.8) mm, rotated rx 0 ry 90 rz 0 deg; joints [-12.093, -27.699, 110.565, -16.141, -82.283, 51.207]
  Set speed (30.0 mm/s)
  Call Extruder(0.280)
  MoveL 7211 to (500.58, 509.32, 14.8) mm, rotated rx 0 ry 90 rz 0 deg; joints [-12.847, -27.802, 111.201, -16.881, -82.818, 51.141]
  Set speed (120.0 mm/s)
  MoveL 7212 to (499.42, 509.32, 14.8) mm, rotated rx 0 ry 90 rz 0 deg; joints [-12.872, -27.824, 111.339, -16.901, -82.93, 51.11]
  Set speed (30.0 mm/s)
  Call Extruder(0.360)
  MoveL 7213 to (490.68, 500.58, 14.8) mm, rotated rx 0 ry 90 rz 0 deg; joints [-12.247, -28.016, 112.607, -16.237, -83.943, 50.738]
  Set speed (120.0 mm/s)
  MoveL 7214 to (490.68, 499.42, 14.8) mm, rotated rx 0 ry 90 rz 0 deg; joints [-12.139, -28.02, 112.637, -16.128, -83.965, 50.722]
  Set speed (30.0 mm/s)
  Call Extruder(0.281)
  MoveL 7215 to (497.52, 492.58, 14.8) mm, rotated rx 0 ry 90 rz 0 deg; joints [-11.373, -27.925, 111.994, -15.374, -83.417, 50.798]
  Set speed (120.0 mm/s)
  MoveL 7216 to (498.28, 491.81, 14.8) mm, rotated rx 0 ry 90 rz 0 deg; joints [-11.288, -27.914, 111.921, -15.291, -83.355, 50.806]
  Set speed (30.0 mm/s)
  Call Extruder(0.047)
  MoveL 7217 to (499.42, 490.68, 14.8) mm, rotated rx 0 ry 90 rz 0 deg; joints [-11.163, -27.898, 111.812, -15.167, -83.263, 50.818]
  Set speed (120.0 mm/s)
  MoveL 7218 to (500.58, 490.68, 14.8) mm, rotated rx 0 ry 90 rz 0 deg; joints [-11.141, -27.876, 111.674, -15.149, -83.149, 50.846]
  Set speed (30.0 mm/s)
  Call Extruder(0.018)
  MoveL 7219 to (501.01, 491.11, 14.8) mm, rotated rx 0 ry 90 rz 0 deg; joints [-11.173, -27.867, 111.612, -15.183, -83.099, 50.863]
  Set speed (120.0 mm/s)
  MoveL 7220 to (502.48, 492.58, 14.8) mm, rotated rx 0 ry 90 rz 0 deg; joints [-11.282, -27.834, 111.401, -15.298, -82.931, 50.922]
  Set speed (30.0 mm/s)
  Call Extruder(0.202)
  MoveL 7221 to (507.39, 497.49, 14.8) mm, rotated rx 0 ry 90 rz 0 deg; joints [-11.639, -27.72, 110.692, -15.678, -82.369, 51.123]
  Set speed (120.0 mm/s)
  MoveL 7222 to (507.76, 497.86, 14.8) mm, rotated rx 0 ry 90 rz 0 deg; joints [-11.666, -27.711, 110.638, -15.707, -82.326, 51.138]
  Set speed (30.0 mm/s)
  Call Extruder(0.064)
  MoveL 7223 to (509.32, 499.42, 14.8) mm, rotated rx 0 ry 90 rz 0 deg; joints [-11.777, -27.673, 110.412, -15.827, -82.148, 51.204]
  Set speed (120.0 mm/s)
  MoveL 7224 to (509.32, 500.58, 14.8) mm, rotated rx 0 ry 90 rz 0 deg; joints [-11.882, -27.668, 110.382, -15.933, -82.129, 51.223]
  Set speed (30.0 mm/s)
  Call Extruder(0.025)
  MoveL 7225 to (508.71, 501.19, 14.8) mm, rotated rx 0 ry 90 rz 0 deg; joints [-11.949, -27.678, 110.44, -15.999, -82.177, 51.218]
  Set speed (120.0 mm/s)
  MoveL 7226 to (507.65, 497.61, 14.8) mm, rotated rx 0 ry 90 rz 0 deg; joints [-11.645, -27.714, 110.658, -15.686, -82.342, 51.131]
  Set speed (1000.0 mm/s)
  MoveL 7227 to (507.65, 495.03, 14.8) mm, rotated rx 0 ry 90 rz 0 deg; joints [-11.411, -27.725, 110.722, -15.447, -82.385, 51.089]
  Set speed (1000.0 mm/s)
  MoveL 7228 to (509.32, 490.68, 14.8) mm, rotated rx 0 ry 90 rz 0 deg; joints [-10.985, -27.708, 110.624, -15.021, -82.293, 51.06]
  Set speed (30.0 mm/s)
  Call Extruder(0.767)
  MoveL 7229 to (490.68, 509.32, 14.8) mm, rotated rx 0 ry 90 rz 0 deg; joints [-13.056, -27.982, 112.375, -17.057, -83.776, 50.87]
  MoveL 7230 to (490.56, 509.44, 14.8) mm, rotated rx 0 ry 90 rz 0 deg; joints [-13.07, -27.984, 112.386, -17.07, -83.785, 50.869]
  Set speed (120.0 mm/s)
  MoveL 7231 to (507.6, 501.4, 14.8) mm, rotated rx 0 ry 90 rz 0 deg; joints [-11.989, -27.699, 110.568, -16.035, -82.281, 51.193]
  Set speed (1000.0 mm/s)
  MoveL 7232 to (507.67, 501.47, 14.8) mm, rotated rx 0 ry 90 rz 0 deg; joints [-11.994, -27.698, 110.558, -16.04, -82.273, 51.196]
  Set speed (15.0 mm/s)
  Call Extruder(0.010)
  MoveL 7233 to (507.67, 501.82, 14.8) mm, rotated rx 0 ry 90 rz 0 deg; joints [-12.025, -27.696, 110.549, -16.073, -82.267, 51.202]
  Call Extruder(0.063)
  MoveL 7234 to (507.67, 503.98, 14.8) mm, rotated rx 0 ry 90 rz 0 deg; joints [-12.22, -27.687, 110.494, -16.271, -82.23, 51.239]
  Call Extruder(0.056)
  MoveL 7235 to (509.6, 503.98, 14.8) mm, rotated rx 0 ry 90 rz 0 deg; joints [-12.183, -27.648, 110.261, -16.241, -82.042, 51.289]
  Call Extruder(0.164)
  MoveL 7236 to (509.6, 509.6, 14.8) mm, rotated rx 0 ry 90 rz 0 deg; joints [-12.688, -27.622, 110.112, -16.756, -81.942, 51.388]
  Call Extruder(0.559)
  MoveL 7237 to (490.4, 509.6, 14.8) mm, rotated rx 0 ry 90 rz 0 deg; joints [-13.088, -27.986, 112.401, -17.088, -83.797, 50.867]
  MoveL 7238 to (490.4, 490.4, 14.8) mm, rotated rx 0 ry 90 rz 0 deg; joints [-11.303, -28.056, 112.891, -15.282, -84.154, 50.588]
  Call Extruder(0.140)
  MoveL 7239 to (495.2, 490.4, 14.8) mm, rotated rx 0 ry 90 rz 0 deg; joints [-11.214, -27.974, 112.321, -15.206, -83.682, 50.709]
  Call Extruder(0.010)
  MoveL 7240 to (495.55, 490.4, 14.8) mm, rotated rx 0 ry 90 rz 0 deg; joints [-11.208, -27.968, 112.28, -15.2, -83.647, 50.717]
  Call Extruder(0.007)
  MoveL 7241 to (495.55, 490.75, 14.8) mm, rotated rx 0 ry 90 rz 0 deg; joints [-11.24, -27.967, 112.272, -15.233, -83.641, 50.722]
  Call Extruder(0.035)
  MoveL 7242 to (495.55, 491.95, 14.8) mm, rotated rx 0 ry 90 rz 0 deg; joints [-11.352, -27.963, 112.243, -15.346, -83.621, 50.739]
  Call Extruder(0.010)
  MoveL 7243 to (495.55, 492.3, 14.8) mm, rotated rx 0 ry 90 rz 0 deg; joints [-11.384, -27.961, 112.235, -15.379, -83.615, 50.745]
  Call Extruder(0.007)
  MoveL 7244 to (495.9, 492.3, 14.8) mm, rotated rx 0 ry 90 rz 0 deg; joints [-11.377, -27.955, 112.193, -15.373, -83.581, 50.753]
  Call Extruder(0.061)
  MoveL 7245 to (498, 492.3, 14.8) mm, rotated rx 0 ry 90 rz 0 deg; joints [-11.338, -27.918, 111.943, -15.341, -83.374, 50.806]
  Call Extruder(0.055)
  MoveL 7246 to (498.01, 490.4, 14.8) mm, rotated rx 0 ry 90 rz 0 deg; joints [-11.163, -27.924, 111.987, -15.162, -83.406, 50.778]
  Call Extruder(0.096)
  MoveL 7247 to (501.29, 490.4, 14.8) mm, rotated rx 0 ry 90 rz 0 deg; joints [-11.103, -27.864, 111.595, -15.113, -83.084, 50.86]
  Call Extruder(0.055)
  MoveL 7248 to (501.29, 492.3, 14.8) mm, rotated rx 0 ry 90 rz 0 deg; joints [-11.278, -27.857, 111.55, -15.29, -83.052, 50.888]
  Call Extruder(0.061)
  MoveL 7249 to (503.38, 492.3, 14.8) mm, rotated rx 0 ry 90 rz 0 deg; joints [-11.24, -27.818, 111.3, -15.258, -82.847, 50.94]
  Call Extruder(0.010)
  MoveL 7250 to (503.73, 492.3, 14.8) mm, rotated rx 0 ry 90 rz 0 deg; joints [-11.233, -27.811, 111.258, -15.253, -82.813, 50.949]
  Call Extruder(0.007)
  MoveL 7251 to (503.73, 491.95, 14.8) mm, rotated rx 0 ry 90 rz 0 deg; joints [-11.201, -27.813, 111.266, -15.221, -82.819, 50.943]
  Call Extruder(0.035)
  MoveL 7252 to (503.73, 490.75, 14.8) mm, rotated rx 0 ry 90 rz 0 deg; joints [-11.091, -27.817, 111.295, -15.109, -82.839, 50.925]
  Call Extruder(0.010)
  MoveL 7253 to (503.73, 490.4, 14.8) mm, rotated rx 0 ry 90 rz 0 deg; joints [-11.059, -27.818, 111.303, -15.076, -82.845, 50.919]
  Call Extruder(0.007)
  MoveL 7254 to (504.08, 490.4, 14.8) mm, rotated rx 0 ry 90 rz 0 deg; joints [-11.053, -27.812, 111.261, -15.071, -82.81, 50.928]
  Call Extruder(0.161)
  MoveL 7255 to (509.6, 490.4, 14.8) mm, rotated rx 0 ry 90 rz 0 deg; joints [-10.955, -27.704, 110.596, -14.992, -82.27, 51.062]
  Call Extruder(0.136)
  MoveL 7256 to (509.6, 495.06, 14.8) mm, rotated rx 0 ry 90 rz 0 deg; joints [-11.377, -27.685, 110.485, -15.421, -82.194, 51.138]
  Call Extruder(0.056)
  MoveL 7257 to (507.67, 495.06, 14.8) mm, rotated rx 0 ry 90 rz 0 deg; joints [-11.413, -27.724, 110.718, -15.45, -82.382, 51.09]
  Call Extruder(0.073)
  MoveL 7258 to (507.67, 497.58, 14.8) mm, rotated rx 0 ry 90 rz 0 deg; joints [-11.642, -27.714, 110.656, -15.683, -82.34, 51.132]
  Call Extruder(0.056)
  MoveL 7259 to (509.6, 497.58, 14.8) mm, rotated rx 0 ry 90 rz 0 deg; joints [-11.606, -27.675, 110.423, -15.653, -82.152, 51.18]
  Call Extruder(0.103)
  MoveL 7260 to (509.6, 501.12, 14.8) mm, rotated rx 0 ry 90 rz 0 deg; joints [-11.925, -27.66, 110.335, -15.979, -82.092, 51.24]
  Call Extruder(0.010)
  MoveL 7261 to (509.6, 501.47, 14.8) mm, rotated rx 0 ry 90 rz 0 deg; joints [-11.957, -27.659, 110.326, -16.011, -82.086, 51.246]
  Call Extruder(0.007)
  MoveL 7262 to (509.25, 501.47, 14.8) mm, rotated rx 0 ry 90 rz 0 deg; joints [-11.964, -27.666, 110.368, -16.016, -82.12, 51.237]
  Call Extruder(0.036)
  MoveL 7263 to (508.02, 501.47, 14.8) mm, rotated rx 0 ry 90 rz 0 deg; joints [-11.987, -27.691, 110.516, -16.035, -82.239, 51.205]
  Call Extruder(0.007)
  MoveL 7264 to (507.67, 501.47, 14.8) mm, rotated rx 0 ry 90 rz 0 deg; joints [-11.994, -27.698, 110.558, -16.04, -82.273, 51.196]
  Set speed (120.0 mm/s)
  MoveL 7265 to (507.67, 501.82, 14.8) mm, rotated rx 0 ry 90 rz 0 deg; joints [-12.025, -27.696, 110.549, -16.073, -82.267, 51.202]
  Set speed (1000.0 mm/s)
  MoveL 7266 to (507.67, 501.87, 14.8) mm, rotated rx 0 ry 90 rz 0 deg; joints [-12.03, -27.696, 110.548, -16.077, -82.266, 51.203]
  Set speed (1000.0 mm/s)
  MoveL 7267 to (506.97, 501.87, 14.8) mm, rotated rx 0 ry 90 rz 0 deg; joints [-12.043, -27.71, 110.632, -16.088, -82.334, 51.185]
  Set speed (1000.0 mm/s)
  MoveL 7268 to (490.68, 490.68, 14.8) mm, rotated rx 0 ry 90 rz 0 deg; joints [-11.324, -28.051, 112.851, -15.304, -84.122, 50.599]
  Set speed (1000.0 mm/s)
  MoveL 7269 to (490.68, 490.68, 14.9) mm, rotated rx 0 ry 90 rz 0 deg; joints [-11.324, -28.061, 112.856, -15.304, -84.116, 50.6]
  Set speed (30.0 mm/s)
  Call Extruder(0.767)
  MoveL 7270 to (509.32, 509.32, 14.9) mm, rotated rx 0 ry 90 rz 0 deg; joints [-12.669, -27.64, 110.158, -16.735, -81.969, 51.377]
  MoveL 7271 to (509.44, 509.44, 14.9) mm, rotated rx 0 ry 90 rz 0 deg; joints [-12.677, -27.637, 110.14, -16.744, -81.955, 51.382]
  Set speed (120.0 mm/s)
  MoveL 7272 to (507.64, 504.06, 14.9) mm, rotated rx 0 ry 90 rz 0 deg; joints [-12.229, -27.697, 110.5, -16.279, -82.226, 51.241]
  Set speed (1000.0 mm/s)
  MoveL 7273 to (507.39, 502.51, 14.9) mm, rotated rx 0 ry 90 rz 0 deg; joints [-12.093, -27.709, 110.571, -16.141, -82.277, 51.208]
  Set speed (30.0 mm/s)
  Call Extruder(0.280)
  MoveL 7274 to (500.58, 509.32, 14.9) mm, rotated rx 0 ry 90 rz 0 deg; joints [-12.847, -27.813, 111.206, -16.881, -82.813, 51.143]
  Set speed (120.0 mm/s)
  MoveL 7275 to (499.42, 509.32, 14.9) mm, rotated rx 0 ry 90 rz 0 deg; joints [-12.872, -27.835, 111.344, -16.901, -82.925, 51.111]
  Set speed (30.0 mm/s)
  Call Extruder(0.360)
  MoveL 7276 to (490.68, 500.58, 14.9) mm, rotated rx 0 ry 90 rz 0 deg; joints [-12.247, -28.027, 112.612, -16.237, -83.938, 50.74]
  Set speed (120.0 mm/s)
  MoveL 7277 to (490.68, 499.42, 14.9) mm, rotated rx 0 ry 90 rz 0 deg; joints [-12.139, -28.031, 112.642, -16.128, -83.96, 50.723]
  Set speed (30.0 mm/s)
  Call Extruder(0.281)
  MoveL 7278 to (497.52, 492.58, 14.9) mm, rotated rx 0 ry 90 rz 0 deg; joints [-11.373, -27.936, 111.999, -15.375, -83.412, 50.8]
  Set speed (120.0 mm/s)
  MoveL 7279 to (498.23, 491.87, 14.9) mm, rotated rx 0 ry 90 rz 0 deg; joints [-11.294, -27.926, 111.932, -15.297, -83.354, 50.807]
  Set speed (30.0 mm/s)
  Call Extruder(0.049)
  MoveL 7280 to (499.42, 490.68, 14.9) mm, rotated rx 0 ry 90 rz 0 deg; joints [-11.163, -27.908, 111.817, -15.167, -83.258, 50.819]
  Set speed (120.0 mm/s)
  MoveL 7281 to (500.58, 490.68, 14.9) mm, rotated rx 0 ry 90 rz 0 deg; joints [-11.142, -27.887, 111.679, -15.15, -83.144, 50.848]
  Set speed (30.0 mm/s)
  Call Extruder(0.020)
  MoveL 7282 to (501.07, 491.17, 14.9) mm, rotated rx 0 ry 90 rz 0 deg; joints [-11.178, -27.876, 111.608, -15.188, -83.087, 50.867]
  Set speed (120.0 mm/s)
  MoveL 7283 to (502.48, 492.58, 14.9) mm, rotated rx 0 ry 90 rz 0 deg; joints [-11.282, -27.844, 111.406, -15.298, -82.926, 50.924]
  Set speed (30.0 mm/s)
  Call Extruder(0.202)
  MoveL 7284 to (507.39, 497.49, 14.9) mm, rotated rx 0 ry 90 rz 0 deg; joints [-11.639, -27.73, 110.697, -15.679, -82.363, 51.125]
  Set speed (120.0 mm/s)
  MoveL 7285 to (507.71, 497.81, 14.9) mm, rotated rx 0 ry 90 rz 0 deg; joints [-11.661, -27.723, 110.651, -15.703, -82.328, 51.138]
  Set speed (30.0 mm/s)
  Call Extruder(0.066)
  MoveL 7286 to (509.32, 499.42, 14.9) mm, rotated rx 0 ry 90 rz 0 deg; joints [-11.777, -27.684, 110.417, -15.827, -82.143, 51.205]
  Set speed (120.0 mm/s)
  MoveL 7287 to (509.32, 500.58, 14.9) mm, rotated rx 0 ry 90 rz 0 deg; joints [-11.882, -27.679, 110.387, -15.933, -82.123, 51.225]
  Set speed (30.0 mm/s)
  Call Extruder(0.027)
  MoveL 7288 to (508.65, 501.25, 14.9) mm, rotated rx 0 ry 90 rz 0 deg; joints [-11.955, -27.689, 110.451, -16.005, -82.177, 51.219]
  Set speed (120.0 mm/s)
  MoveL 7289 to (507.65, 497.55, 14.9) mm, rotated rx 0 ry 90 rz 0 deg; joints [-11.64, -27.725, 110.665, -15.68, -82.338, 51.132]
  Set speed (1000.0 mm/s)
  MoveL 7290 to (507.64, 494.97, 14.9) mm, rotated rx 0 ry 90 rz 0 deg; joints [-11.405, -27.735, 110.728, -15.442, -82.381, 51.09]
  Set speed (1000.0 mm/s)
  MoveL 7291 to (509.32, 490.68, 14.9) mm, rotated rx 0 ry 90 rz 0 deg; joints [-10.985, -27.719, 110.629, -15.021, -82.287, 51.061]
  Set speed (30.0 mm/s)
  Call Extruder(0.767)
  MoveL 7292 to (490.68, 509.32, 14.9) mm, rotated rx 0 ry 90 rz 0 deg; joints [-13.056, -27.993, 112.38, -17.057, -83.771, 50.872]
  MoveL 7293 to (490.56, 509.44, 14.9) mm, rotated rx 0 ry 90 rz 0 deg; joints [-13.07, -27.994, 112.392, -17.071, -83.78, 50.87]
  Set speed (120.0 mm/s)
  MoveL 7294 to (503.87, 492.37, 14.9) mm, rotated rx 0 ry 90 rz 0 deg; joints [-11.237, -27.819, 111.245, -15.258, -82.794, 50.955]
  Set speed (1000.0 mm/s)
  MoveL 7295 to (503.8, 492.3, 14.9) mm, rotated rx 0 ry 90 rz 0 deg; joints [-11.232, -27.821, 111.255, -15.252, -82.802, 50.952]
  Set speed (15.0 mm/s)
  Call Extruder(0.010)
  MoveL 7296 to (503.8, 491.95, 14.9) mm, rotated rx 0 ry 90 rz 0 deg; joints [-11.2, -27.822, 111.264, -15.22, -82.807, 50.946]
  Call Extruder(0.035)
  MoveL 7297 to (503.79, 490.75, 14.9) mm, rotated rx 0 ry 90 rz 0 deg; joints [-11.09, -27.826, 111.292, -15.108, -82.827, 50.928]
  Call Extruder(0.010)
  MoveL 7298 to (503.79, 490.4, 14.9) mm, rotated rx 0 ry 90 rz 0 deg; joints [-11.058, -27.828, 111.3, -15.076, -82.833, 50.922]
  Call Extruder(0.007)
  MoveL 7299 to (504.14, 490.4, 14.9) mm, rotated rx 0 ry 90 rz 0 deg; joints [-11.052, -27.821, 111.258, -15.071, -82.799, 50.931]
  Call Extruder(0.159)
  MoveL 7300 to (509.6, 490.4, 14.9) mm, rotated rx 0 ry 90 rz 0 deg; joints [-10.955, -27.714, 110.601, -14.992, -82.264, 51.064]
  Call Extruder(0.134)
  MoveL 7301 to (509.6, 495, 14.9) mm, rotated rx 0 ry 90 rz 0 deg; joints [-11.372, -27.696, 110.492, -15.416, -82.19, 51.139]
  Call Extruder(0.056)
  MoveL 7302 to (507.67, 495, 14.9) mm, rotated rx 0 ry 90 rz 0 deg; joints [-11.407, -27.735, 110.724, -15.444, -82.378, 51.091]
  Call Extruder(0.073)
  MoveL 7303 to (507.67, 497.52, 14.9) mm, rotated rx 0 ry 90 rz 0 deg; joints [-11.637, -27.724, 110.662, -15.677, -82.335, 51.132]
  Call Extruder(0.056)
  MoveL 7304 to (509.6, 497.53, 14.9) mm, rotated rx 0 ry 90 rz 0 deg; joints [-11.601, -27.686, 110.43, -15.648, -82.148, 51.181]
  Call Extruder(0.106)
  MoveL 7305 to (509.6, 501.18, 14.9) mm, rotated rx 0 ry 90 rz 0 deg; joints [-11.931, -27.67, 110.338, -15.984, -82.086, 51.242]
  Call Extruder(0.010)
  MoveL 7306 to (509.6, 501.53, 14.9) mm, rotated rx 0 ry 90 rz 0 deg; joints [-11.962, -27.669, 110.329, -16.016, -82.08, 51.248]
  Call Extruder(0.007)
  MoveL 7307 to (509.25, 501.53, 14.9) mm, rotated rx 0 ry 90 rz 0 deg; joints [-11.969, -27.676, 110.372, -16.021, -82.114, 51.239]
  Call Extruder(0.036)
  MoveL 7308 to (508.02, 501.52, 14.9) mm, rotated rx 0 ry 90 rz 0 deg; joints [-11.992, -27.701, 110.52, -16.04, -82.233, 51.208]
  Call Extruder(0.010)
  MoveL 7309 to (507.67, 501.52, 14.9) mm, rotated rx 0 ry 90 rz 0 deg; joints [-11.999, -27.708, 110.562, -16.046, -82.267, 51.199]
  Call Extruder(0.007)
  MoveL 7310 to (507.67, 501.87, 14.9) mm, rotated rx 0 ry 90 rz 0 deg; joints [-12.03, -27.706, 110.553, -16.078, -82.261, 51.205]
  Call Extruder(0.063)
  MoveL 7311 to (507.67, 504.03, 14.9) mm, rotated rx 0 ry 90 rz 0 deg; joints [-12.225, -27.697, 110.497, -16.276, -82.223, 51.241]
  Call Extruder(0.056)
  MoveL 7312 to (509.6, 504.03, 14.9) mm, rotated rx 0 ry 90 rz 0 deg; joints [-12.188, -27.658, 110.265, -16.246, -82.036, 51.291]
  Call Extruder(0.162)
  MoveL 7313 to (509.6, 509.6, 14.9) mm, rotated rx 0 ry 90 rz 0 deg; joints [-12.688, -27.633, 110.117, -16.756, -81.937, 51.389]
  Call Extruder(0.559)
  MoveL 7314 to (490.4, 509.6, 14.9) mm, rotated rx 0 ry 90 rz 0 deg; joints [-13.088, -27.996, 112.406, -17.088, -83.792, 50.869]
  MoveL 7315 to (490.4, 490.4, 14.9) mm, rotated rx 0 ry 90 rz 0 deg; joints [-11.303, -28.067, 112.896, -15.282, -84.149, 50.589]
  Call Extruder(0.138)
  MoveL 7316 to (495.15, 490.4, 14.9) mm, rotated rx 0 ry 90 rz 0 deg; joints [-11.215, -27.986, 112.333, -15.207, -83.682, 50.709]
  Call Extruder(0.010)
  MoveL 7317 to (495.5, 490.4, 14.9) mm, rotated rx 0 ry 90 rz 0 deg; joints [-11.209, -27.98, 112.292, -15.201, -83.647, 50.717]
  Call Extruder(0.007)
  MoveL 7318 to (495.5, 490.75, 14.9) mm, rotated rx 0 ry 90 rz 0 deg; joints [-11.241, -27.978, 112.283, -15.234, -83.641, 50.722]
  Call Extruder(0.035)
  MoveL 7319 to (495.49, 491.95, 14.9) mm, rotated rx 0 ry 90 rz 0 deg; joints [-11.353, -27.974, 112.255, -15.347, -83.621, 50.74]
  Call Extruder(0.010)
  MoveL 7320 to (495.49, 492.3, 14.9) mm, rotated rx 0 ry 90 rz 0 deg; joints [-11.385, -27.973, 112.247, -15.38, -83.615, 50.745]
  Call Extruder(0.007)
  MoveL 7321 to (495.84, 492.3, 14.9) mm, rotated rx 0 ry 90 rz 0 deg; joints [-11.379, -27.967, 112.205, -15.374, -83.581, 50.753]
  Call Extruder(0.061)
  MoveL 7322 to (497.95, 492.3, 14.9) mm, rotated rx 0 ry 90 rz 0 deg; joints [-11.339, -27.929, 111.954, -15.342, -83.374, 50.806]
  Call Extruder(0.055)
  MoveL 7323 to (497.95, 490.4, 14.9) mm, rotated rx 0 ry 90 rz 0 deg; joints [-11.164, -27.936, 111.999, -15.163, -83.406, 50.778]
  Call Extruder(0.099)
  MoveL 7324 to (501.35, 490.4, 14.9) mm, rotated rx 0 ry 90 rz 0 deg; joints [-11.102, -27.874, 111.593, -15.112, -83.072, 50.863]
  Call Extruder(0.030)
  MoveL 7325 to (501.35, 491.44, 14.9) mm, rotated rx 0 ry 90 rz 0 deg; joints [-11.197, -27.87, 111.568, -15.209, -83.055, 50.878]
  Call Extruder(0.025)
  MoveL 7326 to (501.36, 492.3, 14.9) mm, rotated rx 0 ry 90 rz 0 deg; joints [-11.277, -27.867, 111.548, -15.289, -83.041, 50.891]
  Call Extruder(0.061)
  MoveL 7327 to (503.44, 492.3, 14.9) mm, rotated rx 0 ry 90 rz 0 deg; joints [-11.238, -27.827, 111.297, -15.258, -82.836, 50.943]
  Call Extruder(0.007)
  MoveL 7328 to (503.8, 492.3, 14.9) mm, rotated rx 0 ry 90 rz 0 deg; joints [-11.232, -27.821, 111.255, -15.252, -82.802, 50.952]
  Set speed (120.0 mm/s)
  MoveL 7329 to (503.8, 491.95, 14.9) mm, rotated rx 0 ry 90 rz 0 deg; joints [-11.2, -27.822, 111.264, -15.22, -82.807, 50.946]
  Set speed (1000.0 mm/s)
  MoveL 7330 to (503.79, 491.9, 14.9) mm, rotated rx 0 ry 90 rz 0 deg; joints [-11.195, -27.822, 111.265, -15.215, -82.808, 50.946]
  Set speed (1000.0 mm/s)
  MoveL 7331 to (504.49, 491.9, 14.9) mm, rotated rx 0 ry 90 rz 0 deg; joints [-11.183, -27.809, 111.181, -15.205, -82.74, 50.963]
  Set speed (1000.0 mm/s)
  MoveL 7332 to (495.47, 492.33, 14.9) mm, rotated rx 0 ry 90 rz 0 deg; joints [-11.388, -27.973, 112.249, -15.383, -83.617, 50.744]
  Set speed (1000.0 mm/s)
  MoveL 7333 to (490.68, 490.68, 14.9) mm, rotated rx 0 ry 90 rz 0 deg; joints [-11.324, -28.061, 112.856, -15.304, -84.116, 50.6]
  Set speed (1000.0 mm/s)
  MoveL 7334 to (490.68, 490.68, 15) mm, rotated rx 0 ry 90 rz 0 deg; joints [-11.324, -28.072, 112.862, -15.304, -84.111, 50.602]
  Set speed (30.0 mm/s)
  Call Extruder(0.767)
  MoveL 7335 to (509.32, 509.32, 15) mm, rotated rx 0 ry 90 rz 0 deg; joints [-12.669, -27.65, 110.163, -16.735, -81.964, 51.378]
  MoveL 7336 to (509.44, 509.44, 15) mm, rotated rx 0 ry 90 rz 0 deg; joints [-12.677, -27.647, 110.145, -16.744, -81.95, 51.384]
  Set speed (120.0 mm/s)
  MoveL 7337 to (507.64, 504.12, 15) mm, rotated rx 0 ry 90 rz 0 deg; joints [-12.234, -27.708, 110.503, -16.285, -82.219, 51.244]
  Set speed (1000.0 mm/s)
  MoveL 7338 to (507.39, 502.51, 15) mm, rotated rx 0 ry 90 rz 0 deg; joints [-12.093, -27.72, 110.576, -16.141, -82.272, 51.21]
  Set speed (30.0 mm/s)
  Call Extruder(0.280)
  MoveL 7339 to (500.58, 509.32, 15) mm, rotated rx 0 ry 90 rz 0 deg; joints [-12.847, -27.823, 111.211, -16.881, -82.808, 51.144]
  Set speed (120.0 mm/s)
  MoveL 7340 to (499.42, 509.32, 15) mm, rotated rx 0 ry 90 rz 0 deg; joints [-12.872, -27.845, 111.349, -16.901, -82.92, 51.113]
  Set speed (30.0 mm/s)
  Call Extruder(0.360)
  MoveL 7341 to (490.68, 500.58, 15) mm, rotated rx 0 ry 90 rz 0 deg; joints [-12.247, -28.037, 112.617, -16.237, -83.933, 50.742]
  Set speed (120.0 mm/s)
  MoveL 7342 to (490.68, 499.42, 15) mm, rotated rx 0 ry 90 rz 0 deg; joints [-12.139, -28.041, 112.647, -16.128, -83.954, 50.725]
  Set speed (30.0 mm/s)
  Call Extruder(0.281)
  MoveL 7343 to (497.52, 492.58, 15) mm, rotated rx 0 ry 90 rz 0 deg; joints [-11.373, -27.947, 112.004, -15.375, -83.407, 50.801]
  Set speed (120.0 mm/s)
  MoveL 7344 to (498.17, 491.93, 15) mm, rotated rx 0 ry 90 rz 0 deg; joints [-11.301, -27.937, 111.942, -15.303, -83.354, 50.808]
  Set speed (30.0 mm/s)
  Call Extruder(0.051)
  MoveL 7345 to (499.42, 490.68, 15) mm, rotated rx 0 ry 90 rz 0 deg; joints [-11.163, -27.919, 111.823, -15.167, -83.252, 50.82]
  Set speed (120.0 mm/s)
  MoveL 7346 to (500.58, 490.68, 15) mm, rotated rx 0 ry 90 rz 0 deg; joints [-11.141, -27.898, 111.684, -15.15, -83.138, 50.849]
  Set speed (30.0 mm/s)
  Call Extruder(0.023)
  MoveL 7347 to (501.14, 491.24, 15) mm, rotated rx 0 ry 90 rz 0 deg; joints [-11.183, -27.885, 111.604, -15.193, -83.075, 50.871]
  Set speed (120.0 mm/s)
  MoveL 7348 to (502.48, 492.58, 15) mm, rotated rx 0 ry 90 rz 0 deg; joints [-11.282, -27.855, 111.411, -15.298, -82.92, 50.925]
  Set speed (30.0 mm/s)
  Call Extruder(0.202)
  MoveL 7349 to (507.39, 497.5, 15) mm, rotated rx 0 ry 90 rz 0 deg; joints [-11.639, -27.741, 110.702, -15.679, -82.358, 51.126]
  Set speed (120.0 mm/s)
  MoveL 7350 to (507.65, 497.75, 15) mm, rotated rx 0 ry 90 rz 0 deg; joints [-11.657, -27.735, 110.665, -15.698, -82.329, 51.137]
  Set speed (30.0 mm/s)
  Call Extruder(0.069)
  MoveL 7351 to (509.32, 499.42, 15) mm, rotated rx 0 ry 90 rz 0 deg; joints [-11.777, -27.694, 110.422, -15.827, -82.138, 51.207]
  Set speed (120.0 mm/s)
  MoveL 7352 to (509.32, 500.58, 15) mm, rotated rx 0 ry 90 rz 0 deg; joints [-11.882, -27.689, 110.392, -15.934, -82.118, 51.226]
  Set speed (30.0 mm/s)
  Call Extruder(0.030)
  MoveL 7353 to (508.6, 501.3, 15) mm, rotated rx 0 ry 90 rz 0 deg; joints [-11.961, -27.701, 110.461, -16.011, -82.176, 51.22]
  Set speed (120.0 mm/s)
  MoveL 7354 to (507.65, 497.5, 15) mm, rotated rx 0 ry 90 rz 0 deg; joints [-11.634, -27.736, 110.671, -15.675, -82.333, 51.132]
  Set speed (1000.0 mm/s)
  MoveL 7355 to (507.64, 494.91, 15) mm, rotated rx 0 ry 90 rz 0 deg; joints [-11.4, -27.746, 110.735, -15.437, -82.377, 51.09]
  Set speed (1000.0 mm/s)
  MoveL 7356 to (509.32, 490.68, 15) mm, rotated rx 0 ry 90 rz 0 deg; joints [-10.985, -27.729, 110.634, -15.022, -82.282, 51.063]
  Set speed (30.0 mm/s)
  Call Extruder(0.767)
  MoveL 7357 to (490.68, 509.32, 15) mm, rotated rx 0 ry 90 rz 0 deg; joints [-13.056, -28.003, 112.386, -17.057, -83.765, 50.874]
  MoveL 7358 to (490.56, 509.44, 15) mm, rotated rx 0 ry 90 rz 0 deg; joints [-13.07, -28.005, 112.397, -17.071, -83.775, 50.872]
  Set speed (120.0 mm/s)
  MoveL 7359 to (503.93, 492.37, 15) mm, rotated rx 0 ry 90 rz 0 deg; joints [-11.236, -27.828, 111.243, -15.257, -82.782, 50.958]
  Set speed (1000.0 mm/s)
  MoveL 7360 to (503.86, 492.3, 15) mm, rotated rx 0 ry 90 rz 0 deg; joints [-11.231, -27.83, 111.253, -15.252, -82.79, 50.955]
  Set speed (15.0 mm/s)
  Call Extruder(0.010)
  MoveL 7361 to (503.86, 491.95, 15) mm, rotated rx 0 ry 90 rz 0 deg; joints [-11.199, -27.831, 111.261, -15.219, -82.796, 50.949]
  Call Extruder(0.035)
  MoveL 7362 to (503.86, 490.75, 15) mm, rotated rx 0 ry 90 rz 0 deg; joints [-11.089, -27.836, 111.29, -15.108, -82.816, 50.931]
  Call Extruder(0.010)
  MoveL 7363 to (503.86, 490.4, 15) mm, rotated rx 0 ry 90 rz 0 deg; joints [-11.057, -27.837, 111.298, -15.075, -82.822, 50.925]
  Call Extruder(0.007)
  MoveL 7364 to (504.21, 490.4, 15) mm, rotated rx 0 ry 90 rz 0 deg; joints [-11.051, -27.83, 111.256, -15.07, -82.787, 50.934]
  Call Extruder(0.157)
  MoveL 7365 to (509.6, 490.4, 15) mm, rotated rx 0 ry 90 rz 0 deg; joints [-10.955, -27.725, 110.607, -14.992, -82.259, 51.065]
  Call Extruder(0.132)
  MoveL 7366 to (509.6, 494.94, 15) mm, rotated rx 0 ry 90 rz 0 deg; joints [-11.367, -27.707, 110.499, -15.41, -82.186, 51.139]
  Call Extruder(0.056)
  MoveL 7367 to (507.67, 494.94, 15) mm, rotated rx 0 ry 90 rz 0 deg; joints [-11.402, -27.745, 110.731, -15.439, -82.374, 51.091]
  Call Extruder(0.074)
  MoveL 7368 to (507.67, 497.47, 15) mm, rotated rx 0 ry 90 rz 0 deg; joints [-11.631, -27.735, 110.669, -15.672, -82.331, 51.133]
  Call Extruder(0.056)
  MoveL 7369 to (509.6, 497.47, 15) mm, rotated rx 0 ry 90 rz 0 deg; joints [-11.595, -27.697, 110.437, -15.643, -82.144, 51.181]
  Call Extruder(0.110)
  MoveL 7370 to (509.6, 501.23, 15) mm, rotated rx 0 ry 90 rz 0 deg; joints [-11.936, -27.681, 110.342, -15.989, -82.08, 51.245]
  Call Extruder(0.010)
  MoveL 7371 to (509.6, 501.58, 15) mm, rotated rx 0 ry 90 rz 0 deg; joints [-11.967, -27.679, 110.333, -16.021, -82.074, 51.251]
  Call Extruder(0.007)
  MoveL 7372 to (509.25, 501.58, 15) mm, rotated rx 0 ry 90 rz 0 deg; joints [-11.974, -27.686, 110.375, -16.027, -82.108, 51.242]
  Call Extruder(0.036)
  MoveL 7373 to (508.02, 501.58, 15) mm, rotated rx 0 ry 90 rz 0 deg; joints [-11.997, -27.711, 110.523, -16.046, -82.227, 51.21]
  Call Extruder(0.010)
  MoveL 7374 to (507.67, 501.58, 15) mm, rotated rx 0 ry 90 rz 0 deg; joints [-12.004, -27.718, 110.565, -16.051, -82.261, 51.201]
  Call Extruder(0.007)
  MoveL 7375 to (507.67, 501.93, 15) mm, rotated rx 0 ry 90 rz 0 deg; joints [-12.036, -27.717, 110.556, -16.083, -82.255, 51.207]
  Call Extruder(0.063)
  MoveL 7376 to (507.67, 504.09, 15) mm, rotated rx 0 ry 90 rz 0 deg; joints [-12.231, -27.707, 110.501, -16.282, -82.217, 51.244]
  Call Extruder(0.056)
  MoveL 7377 to (509.6, 504.09, 15) mm, rotated rx 0 ry 90 rz 0 deg; joints [-12.193, -27.668, 110.268, -16.252, -82.03, 51.294]
  Call Extruder(0.160)
  MoveL 7378 to (509.6, 509.6, 15) mm, rotated rx 0 ry 90 rz 0 deg; joints [-12.688, -27.643, 110.122, -16.756, -81.932, 51.391]
  Call Extruder(0.559)
  MoveL 7379 to (490.4, 509.6, 15) mm, rotated rx 0 ry 90 rz 0 deg; joints [-13.088, -28.007, 112.411, -17.088, -83.787, 50.87]
  MoveL 7380 to (490.4, 490.4, 15) mm, rotated rx 0 ry 90 rz 0 deg; joints [-11.303, -28.078, 112.901, -15.282, -84.143, 50.591]
  Call Extruder(0.136)
  MoveL 7381 to (495.09, 490.4, 15) mm, rotated rx 0 ry 90 rz 0 deg; joints [-11.216, -27.997, 112.345, -15.208, -83.682, 50.709]
  Call Extruder(0.010)
  MoveL 7382 to (495.44, 490.4, 15) mm, rotated rx 0 ry 90 rz 0 deg; joints [-11.21, -27.991, 112.304, -15.202, -83.648, 50.717]
  Call Extruder(0.007)
  MoveL 7383 to (495.44, 490.75, 15) mm, rotated rx 0 ry 90 rz 0 deg; joints [-11.242, -27.99, 112.295, -15.235, -83.642, 50.722]
  Call Extruder(0.035)
  MoveL 7384 to (495.44, 491.95, 15) mm, rotated rx 0 ry 90 rz 0 deg; joints [-11.354, -27.986, 112.267, -15.348, -83.622, 50.74]
  Call Extruder(0.010)
  MoveL 7385 to (495.44, 492.3, 15) mm, rotated rx 0 ry 90 rz 0 deg; joints [-11.386, -27.985, 112.259, -15.381, -83.616, 50.745]
  Call Extruder(0.007)
  MoveL 7386 to (495.79, 492.3, 15) mm, rotated rx 0 ry 90 rz 0 deg; joints [-11.38, -27.978, 112.217, -15.376, -83.581, 50.753]
  Call Extruder(0.061)
  MoveL 7387 to (497.89, 492.3, 15) mm, rotated rx 0 ry 90 rz 0 deg; joints [-11.341, -27.941, 111.966, -15.343, -83.375, 50.806]
  Call Extruder(0.055)
  MoveL 7388 to (497.89, 490.4, 15) mm, rotated rx 0 ry 90 rz 0 deg; joints [-11.165, -27.948, 112.011, -15.165, -83.407, 50.779]
  Call Extruder(0.102)
  MoveL 7389 to (501.42, 490.4, 15) mm, rotated rx 0 ry 90 rz 0 deg; joints [-11.101, -27.883, 111.59, -15.111, -83.061, 50.866]
  Call Extruder(0.031)
  MoveL 7390 to (501.42, 491.48, 15) mm, rotated rx 0 ry 90 rz 0 deg; joints [-11.2, -27.879, 111.565, -15.212, -83.043, 50.882]
  Call Extruder(0.024)
  MoveL 7391 to (501.42, 492.3, 15) mm, rotated rx 0 ry 90 rz 0 deg; joints [-11.275, -27.876, 111.545, -15.288, -83.029, 50.894]
  Call Extruder(0.061)
  MoveL 7392 to (503.51, 492.3, 15) mm, rotated rx 0 ry 90 rz 0 deg; joints [-11.237, -27.837, 111.295, -15.257, -82.824, 50.946]
  Call Extruder(0.007)
  MoveL 7393 to (503.86, 492.3, 15) mm, rotated rx 0 ry 90 rz 0 deg; joints [-11.231, -27.83, 111.253, -15.252, -82.79, 50.955]
  Set speed (120.0 mm/s)
  MoveL 7394 to (503.86, 491.95, 15) mm, rotated rx 0 ry 90 rz 0 deg; joints [-11.199, -27.831, 111.261, -15.219, -82.796, 50.949]
  Set speed (1000.0 mm/s)
  MoveL 7395 to (503.86, 491.9, 15) mm, rotated rx 0 ry 90 rz 0 deg; joints [-11.194, -27.831, 111.262, -15.214, -82.797, 50.949]
  Set speed (1000.0 mm/s)
  MoveL 7396 to (504.56, 491.9, 15) mm, rotated rx 0 ry 90 rz 0 deg; joints [-11.182, -27.818, 111.178, -15.204, -82.728, 50.966]
  Set speed (1000.0 mm/s)
  MoveL 7397 to (495.41, 492.33, 15) mm, rotated rx 0 ry 90 rz 0 deg; joints [-11.389, -27.985, 112.261, -15.384, -83.618, 50.744]
  Set speed (1000.0 mm/s)
  MoveL 7398 to (490.68, 490.68, 15) mm, rotated rx 0 ry 90 rz 0 deg; joints [-11.324, -28.072, 112.862, -15.304, -84.111, 50.602]
  Set speed (1000.0 mm/s)
  MoveL 7399 to (490.68, 490.68, 15.1) mm, rotated rx 0 ry 90 rz 0 deg; joints [-11.324, -28.083, 112.867, -15.304, -84.106, 50.603]
  Set speed (30.0 mm/s)
  Call Extruder(0.767)
  MoveL 7400 to (509.32, 509.32, 15.1) mm, rotated rx 0 ry 90 rz 0 deg; joints [-12.669, -27.661, 110.168, -16.735, -81.959, 51.38]
  MoveL 7401 to (509.44, 509.44, 15.1) mm, rotated rx 0 ry 90 rz 0 deg; joints [-12.677, -27.658, 110.15, -16.744, -81.945, 51.385]
  Set speed (120.0 mm/s)
  MoveL 7402 to (507.64, 504.17, 15.1) mm, rotated rx 0 ry 90 rz 0 deg; joints [-12.239, -27.718, 110.507, -16.29, -82.213, 51.246]
  Set speed (1000.0 mm/s)
  MoveL 7403 to (507.39, 502.51, 15.1) mm, rotated rx 0 ry 90 rz 0 deg; joints [-12.093, -27.73, 110.58, -16.141, -82.267, 51.211]
  Set speed (30.0 mm/s)
  Call Extruder(0.280)
  MoveL 7404 to (500.58, 509.32, 15.1) mm, rotated rx 0 ry 90 rz 0 deg; joints [-12.847, -27.834, 111.216, -16.881, -82.803, 51.146]
  Set speed (120.0 mm/s)
  MoveL 7405 to (499.42, 509.32, 15.1) mm, rotated rx 0 ry 90 rz 0 deg; joints [-12.872, -27.856, 111.354, -16.901, -82.915, 51.115]
  Set speed (30.0 mm/s)
  Call Extruder(0.360)
  MoveL 7406 to (490.68, 500.58, 15.1) mm, rotated rx 0 ry 90 rz 0 deg; joints [-12.247, -28.048, 112.622, -16.237, -83.928, 50.743]
  Set speed (120.0 mm/s)
  MoveL 7407 to (490.68, 499.42, 15.1) mm, rotated rx 0 ry 90 rz 0 deg; joints [-12.139, -28.052, 112.652, -16.128, -83.949, 50.726]
  Set speed (30.0 mm/s)
  Call Extruder(0.281)
  MoveL 7408 to (497.52, 492.58, 15.1) mm, rotated rx 0 ry 90 rz 0 deg; joints [-11.373, -27.957, 112.01, -15.375, -83.401, 50.802]
  Set speed (120.0 mm/s)
  MoveL 7409 to (498.11, 491.99, 15.1) mm, rotated rx 0 ry 90 rz 0 deg; joints [-11.307, -27.949, 111.953, -15.31, -83.353, 50.809]
  Set speed (30.0 mm/s)
  Call Extruder(0.054)
  MoveL 7410 to (499.42, 490.68, 15.1) mm, rotated rx 0 ry 90 rz 0 deg; joints [-11.163, -27.929, 111.828, -15.168, -83.247, 50.822]
  Set speed (120.0 mm/s)
  MoveL 7411 to (500.58, 490.68, 15.1) mm, rotated rx 0 ry 90 rz 0 deg; joints [-11.142, -27.908, 111.689, -15.15, -83.133, 50.851]
  Set speed (30.0 mm/s)
  Call Extruder(0.025)
  MoveL 7412 to (501.2, 491.3, 15.1) mm, rotated rx 0 ry 90 rz 0 deg; joints [-11.187, -27.894, 111.6, -15.198, -83.062, 50.875]
  Set speed (120.0 mm/s)
  MoveL 7413 to (502.48, 492.58, 15.1) mm, rotated rx 0 ry 90 rz 0 deg; joints [-11.282, -27.866, 111.416, -15.298, -82.915, 50.926]
  Set speed (30.0 mm/s)
  Call Extruder(0.202)
  MoveL 7414 to (507.39, 497.5, 15.1) mm, rotated rx 0 ry 90 rz 0 deg; joints [-11.639, -27.751, 110.707, -15.679, -82.353, 51.128]
  Set speed (120.0 mm/s)
  MoveL 7415 to (507.59, 497.69, 15.1) mm, rotated rx 0 ry 90 rz 0 deg; joints [-11.653, -27.746, 110.679, -15.694, -82.331, 51.136]
  Set speed (30.0 mm/s)
  Call Extruder(0.071)
  MoveL 7416 to (509.32, 499.42, 15.1) mm, rotated rx 0 ry 90 rz 0 deg; joints [-11.777, -27.705, 110.427, -15.827, -82.133, 51.208]
  Set speed (120.0 mm/s)
  MoveL 7417 to (509.32, 500.58, 15.1) mm, rotated rx 0 ry 90 rz 0 deg; joints [-11.882, -27.7, 110.398, -15.934, -82.113, 51.228]
  Set speed (30.0 mm/s)
  Call Extruder(0.032)
  MoveL 7418 to (508.54, 501.36, 15.1) mm, rotated rx 0 ry 90 rz 0 deg; joints [-11.967, -27.712, 110.471, -16.017, -82.175, 51.221]
  Set speed (120.0 mm/s)
  MoveL 7419 to (507.65, 497.44, 15.1) mm, rotated rx 0 ry 90 rz 0 deg; joints [-11.629, -27.746, 110.678, -15.67, -82.329, 51.133]
  Set speed (1000.0 mm/s)
  MoveL 7420 to (507.64, 494.85, 15.1) mm, rotated rx 0 ry 90 rz 0 deg; joints [-11.394, -27.757, 110.741, -15.432, -82.373, 51.091]
  Set speed (1000.0 mm/s)
  MoveL 7421 to (509.32, 490.68, 15.1) mm, rotated rx 0 ry 90 rz 0 deg; joints [-10.985, -27.74, 110.639, -15.022, -82.277, 51.064]
  Set speed (30.0 mm/s)
  Call Extruder(0.767)
  MoveL 7422 to (490.68, 509.32, 15.1) mm, rotated rx 0 ry 90 rz 0 deg; joints [-13.056, -28.014, 112.391, -17.057, -83.76, 50.875]
  MoveL 7423 to (490.56, 509.44, 15.1) mm, rotated rx 0 ry 90 rz 0 deg; joints [-13.07, -28.016, 112.402, -17.071, -83.77, 50.874]
  Set speed (120.0 mm/s)
  MoveL 7424 to (503.99, 492.37, 15.1) mm, rotated rx 0 ry 90 rz 0 deg; joints [-11.235, -27.838, 111.24, -15.256, -82.771, 50.961]
  Set speed (1000.0 mm/s)
  MoveL 7425 to (503.92, 492.3, 15.1) mm, rotated rx 0 ry 90 rz 0 deg; joints [-11.23, -27.839, 111.25, -15.251, -82.779, 50.958]
  Set speed (15.0 mm/s)
  Call Extruder(0.010)
  MoveL 7426 to (503.92, 491.95, 15.1) mm, rotated rx 0 ry 90 rz 0 deg; joints [-11.198, -27.841, 111.259, -15.218, -82.785, 50.952]
  Call Extruder(0.035)
  MoveL 7427 to (503.92, 490.75, 15.1) mm, rotated rx 0 ry 90 rz 0 deg; joints [-11.088, -27.845, 111.287, -15.107, -82.804, 50.934]
  Call Extruder(0.010)
  MoveL 7428 to (503.92, 490.4, 15.1) mm, rotated rx 0 ry 90 rz 0 deg; joints [-11.056, -27.846, 111.295, -15.074, -82.81, 50.928]
  Call Extruder(0.007)
  MoveL 7429 to (504.27, 490.4, 15.1) mm, rotated rx 0 ry 90 rz 0 deg; joints [-11.049, -27.84, 111.253, -15.069, -82.776, 50.937]
  Call Extruder(0.155)
  MoveL 7430 to (509.6, 490.4, 15.1) mm, rotated rx 0 ry 90 rz 0 deg; joints [-10.955, -27.735, 110.612, -14.992, -82.254, 51.067]
  Call Extruder(0.130)
  MoveL 7431 to (509.6, 494.88, 15.1) mm, rotated rx 0 ry 90 rz 0 deg; joints [-11.361, -27.718, 110.505, -15.405, -82.182, 51.139]
  Call Extruder(0.056)
  MoveL 7432 to (507.67, 494.88, 15.1) mm, rotated rx 0 ry 90 rz 0 deg; joints [-11.396, -27.756, 110.737, -15.434, -82.369, 51.092]
  Call Extruder(0.074)
  MoveL 7433 to (507.67, 497.41, 15.1) mm, rotated rx 0 ry 90 rz 0 deg; joints [-11.626, -27.746, 110.675, -15.667, -82.327, 51.133]
  Call Extruder(0.056)
  MoveL 7434 to (509.6, 497.41, 15.1) mm, rotated rx 0 ry 90 rz 0 deg; joints [-11.59, -27.707, 110.443, -15.638, -82.139, 51.181]
  Call Extruder(0.113)
  MoveL 7435 to (509.6, 501.29, 15.1) mm, rotated rx 0 ry 90 rz 0 deg; joints [-11.941, -27.691, 110.346, -15.995, -82.074, 51.247]
  Call Extruder(0.010)
  MoveL 7436 to (509.6, 501.64, 15.1) mm, rotated rx 0 ry 90 rz 0 deg; joints [-11.972, -27.689, 110.337, -16.027, -82.068, 51.253]
  Call Extruder(0.007)
  MoveL 7437 to (509.25, 501.64, 15.1) mm, rotated rx 0 ry 90 rz 0 deg; joints [-11.979, -27.696, 110.379, -16.032, -82.102, 51.244]
  Call Extruder(0.036)
  MoveL 7438 to (508.02, 501.64, 15.1) mm, rotated rx 0 ry 90 rz 0 deg; joints [-12.002, -27.721, 110.527, -16.051, -82.221, 51.213]
  Call Extruder(0.010)
  MoveL 7439 to (507.67, 501.63, 15.1) mm, rotated rx 0 ry 90 rz 0 deg; joints [-12.009, -27.728, 110.569, -16.056, -82.255, 51.204]
  Call Extruder(0.007)
  MoveL 7440 to (507.67, 501.99, 15.1) mm, rotated rx 0 ry 90 rz 0 deg; joints [-12.04, -27.727, 110.56, -16.089, -82.249, 51.209]
  Call Extruder(0.063)
  MoveL 7441 to (507.67, 504.15, 15.1) mm, rotated rx 0 ry 90 rz 0 deg; joints [-12.236, -27.717, 110.504, -16.287, -82.211, 51.246]
  Call Extruder(0.056)
  MoveL 7442 to (509.6, 504.15, 15.1) mm, rotated rx 0 ry 90 rz 0 deg; joints [-12.198, -27.678, 110.272, -16.257, -82.024, 51.296]
  Call Extruder(0.159)
  MoveL 7443 to (509.6, 509.6, 15.1) mm, rotated rx 0 ry 90 rz 0 deg; joints [-12.688, -27.654, 110.127, -16.756, -81.927, 51.393]
  Call Extruder(0.559)
  MoveL 7444 to (490.4, 509.6, 15.1) mm, rotated rx 0 ry 90 rz 0 deg; joints [-13.088, -28.018, 112.416, -17.089, -83.782, 50.872]
  MoveL 7445 to (490.4, 490.4, 15.1) mm, rotated rx 0 ry 90 rz 0 deg; joints [-11.303, -28.088, 112.906, -15.282, -84.138, 50.592]
  Call Extruder(0.135)
  MoveL 7446 to (495.03, 490.4, 15.1) mm, rotated rx 0 ry 90 rz 0 deg; joints [-11.217, -28.009, 112.357, -15.209, -83.682, 50.709]
  Call Extruder(0.010)
  MoveL 7447 to (495.38, 490.4, 15.1) mm, rotated rx 0 ry 90 rz 0 deg; joints [-11.211, -28.003, 112.315, -15.203, -83.648, 50.717]
  Call Extruder(0.007)
  MoveL 7448 to (495.38, 490.75, 15.1) mm, rotated rx 0 ry 90 rz 0 deg; joints [-11.243, -28.002, 112.307, -15.236, -83.642, 50.722]
  Call Extruder(0.035)
  MoveL 7449 to (495.38, 491.95, 15.1) mm, rotated rx 0 ry 90 rz 0 deg; joints [-11.355, -27.998, 112.279, -15.349, -83.622, 50.74]
  Call Extruder(0.010)
  MoveL 7450 to (495.38, 492.3, 15.1) mm, rotated rx 0 ry 90 rz 0 deg; joints [-11.387, -27.996, 112.27, -15.382, -83.616, 50.745]
  Call Extruder(0.007)
  MoveL 7451 to (495.73, 492.3, 15.1) mm, rotated rx 0 ry 90 rz 0 deg; joints [-11.381, -27.99, 112.229, -15.377, -83.581, 50.753]
  Call Extruder(0.061)
  MoveL 7452 to (497.83, 492.3, 15.1) mm, rotated rx 0 ry 90 rz 0 deg; joints [-11.342, -27.952, 111.978, -15.344, -83.375, 50.806]
  Call Extruder(0.055)
  MoveL 7453 to (497.84, 490.4, 15.1) mm, rotated rx 0 ry 90 rz 0 deg; joints [-11.166, -27.959, 112.023, -15.166, -83.407, 50.779]
  Call Extruder(0.106)
  MoveL 7454 to (501.48, 490.4, 15.1) mm, rotated rx 0 ry 90 rz 0 deg; joints [-11.1, -27.892, 111.588, -15.11, -83.05, 50.869]
  Call Extruder(0.033)
  MoveL 7455 to (501.48, 491.52, 15.1) mm, rotated rx 0 ry 90 rz 0 deg; joints [-11.202, -27.888, 111.561, -15.215, -83.031, 50.885]
  Call Extruder(0.023)
  MoveL 7456 to (501.48, 492.3, 15.1) mm, rotated rx 0 ry 90 rz 0 deg; joints [-11.274, -27.885, 111.542, -15.288, -83.017, 50.897]
  Call Extruder(0.061)
  MoveL 7457 to (503.57, 492.3, 15.1) mm, rotated rx 0 ry 90 rz 0 deg; joints [-11.236, -27.846, 111.292, -15.256, -82.813, 50.949]
  Call Extruder(0.007)
  MoveL 7458 to (503.92, 492.3, 15.1) mm, rotated rx 0 ry 90 rz 0 deg; joints [-11.23, -27.839, 111.25, -15.251, -82.779, 50.958]
  Set speed (120.0 mm/s)
  MoveL 7459 to (503.92, 491.95, 15.1) mm, rotated rx 0 ry 90 rz 0 deg; joints [-11.198, -27.841, 111.259, -15.218, -82.785, 50.952]
  Set speed (1000.0 mm/s)
  MoveL 7460 to (503.92, 491.9, 15.1) mm, rotated rx 0 ry 90 rz 0 deg; joints [-11.193, -27.841, 111.26, -15.214, -82.785, 50.952]
  Set speed (1000.0 mm/s)
  MoveL 7461 to (504.62, 491.9, 15.1) mm, rotated rx 0 ry 90 rz 0 deg; joints [-11.18, -27.827, 111.176, -15.203, -82.717, 50.969]
  Set speed (1000.0 mm/s)
  MoveL 7462 to (495.35, 492.33, 15.1) mm, rotated rx 0 ry 90 rz 0 deg; joints [-11.39, -27.997, 112.273, -15.385, -83.618, 50.744]
  Set speed (1000.0 mm/s)
  MoveL 7463 to (490.68, 490.68, 15.1) mm, rotated rx 0 ry 90 rz 0 deg; joints [-11.324, -28.083, 112.867, -15.304, -84.106, 50.603]
  Set speed (1000.0 mm/s)
  MoveL 7464 to (490.68, 490.68, 15.2) mm, rotated rx 0 ry 90 rz 0 deg; joints [-11.324, -28.094, 112.872, -15.304, -84.1, 50.605]
  Set speed (30.0 mm/s)
  Call Extruder(0.767)
  MoveL 7465 to (509.32, 509.32, 15.2) mm, rotated rx 0 ry 90 rz 0 deg; joints [-12.669, -27.671, 110.173, -16.735, -81.954, 51.382]
  MoveL 7466 to (509.44, 509.44, 15.2) mm, rotated rx 0 ry 90 rz 0 deg; joints [-12.677, -27.668, 110.155, -16.745, -81.94, 51.387]
  Set speed (120.0 mm/s)
  MoveL 7467 to (507.64, 504.23, 15.2) mm, rotated rx 0 ry 90 rz 0 deg; joints [-12.244, -27.728, 110.511, -16.296, -82.207, 51.248]
  Set speed (1000.0 mm/s)
  MoveL 7468 to (507.39, 502.51, 15.2) mm, rotated rx 0 ry 90 rz 0 deg; joints [-12.093, -27.741, 110.586, -16.141, -82.262, 51.213]
  Set speed (30.0 mm/s)
  Call Extruder(0.280)
  MoveL 7469 to (500.58, 509.32, 15.2) mm, rotated rx 0 ry 90 rz 0 deg; joints [-12.847, -27.844, 111.221, -16.882, -82.797, 51.148]
  Set speed (120.0 mm/s)
  MoveL 7470 to (499.42, 509.32, 15.2) mm, rotated rx 0 ry 90 rz 0 deg; joints [-12.872, -27.866, 111.359, -16.902, -82.909, 51.116]
  Set speed (30.0 mm/s)
  Call Extruder(0.360)
  MoveL 7471 to (490.68, 500.58, 15.2) mm, rotated rx 0 ry 90 rz 0 deg; joints [-12.247, -28.059, 112.628, -16.238, -83.922, 50.745]
  Set speed (120.0 mm/s)
  MoveL 7472 to (490.68, 499.42, 15.2) mm, rotated rx 0 ry 90 rz 0 deg; joints [-12.139, -28.063, 112.657, -16.128, -83.944, 50.728]
  Set speed (30.0 mm/s)
  Call Extruder(0.281)
  MoveL 7473 to (497.51, 492.58, 15.2) mm, rotated rx 0 ry 90 rz 0 deg; joints [-11.373, -27.968, 112.015, -15.375, -83.396, 50.804]
  Set speed (120.0 mm/s)
  MoveL 7474 to (498.06, 492.04, 15.2) mm, rotated rx 0 ry 90 rz 0 deg; joints [-11.313, -27.96, 111.963, -15.316, -83.352, 50.81]
  Set speed (30.0 mm/s)
  Call Extruder(0.056)
  MoveL 7475 to (499.42, 490.68, 15.2) mm, rotated rx 0 ry 90 rz 0 deg; joints [-11.163, -27.94, 111.833, -15.168, -83.242, 50.823]
  Set speed (120.0 mm/s)
  MoveL 7476 to (500.58, 490.68, 15.2) mm, rotated rx 0 ry 90 rz 0 deg; joints [-11.141, -27.919, 111.694, -15.15, -83.128, 50.852]
  Set speed (30.0 mm/s)
  Call Extruder(0.028)
  MoveL 7477 to (501.26, 491.36, 15.2) mm, rotated rx 0 ry 90 rz 0 deg; joints [-11.192, -27.904, 111.596, -15.204, -83.049, 50.879]
  Set speed (120.0 mm/s)
  MoveL 7478 to (502.48, 492.58, 15.2) mm, rotated rx 0 ry 90 rz 0 deg; joints [-11.282, -27.876, 111.421, -15.299, -82.91, 50.928]
  Set speed (30.0 mm/s)
  Call Extruder(0.202)
  MoveL 7479 to (507.4, 497.5, 15.2) mm, rotated rx 0 ry 90 rz 0 deg; joints [-11.639, -27.762, 110.712, -15.679, -82.347, 51.129]
  Set speed (120.0 mm/s)
  MoveL 7480 to (507.53, 497.63, 15.2) mm, rotated rx 0 ry 90 rz 0 deg; joints [-11.649, -27.758, 110.692, -15.69, -82.332, 51.135]
  Set speed (30.0 mm/s)
  Call Extruder(0.074)
  MoveL 7481 to (509.32, 499.42, 15.2) mm, rotated rx 0 ry 90 rz 0 deg; joints [-11.777, -27.715, 110.432, -15.827, -82.128, 51.21]
  Set speed (120.0 mm/s)
  MoveL 7482 to (509.32, 500.58, 15.2) mm, rotated rx 0 ry 90 rz 0 deg; joints [-11.882, -27.71, 110.403, -15.934, -82.108, 51.229]
  Set speed (30.0 mm/s)
  Call Extruder(0.034)
  MoveL 7483 to (508.49, 501.41, 15.2) mm, rotated rx 0 ry 90 rz 0 deg; joints [-11.973, -27.723, 110.482, -16.023, -82.174, 51.222]
  Set speed (120.0 mm/s)
  MoveL 7484 to (507.65, 497.38, 15.2) mm, rotated rx 0 ry 90 rz 0 deg; joints [-11.624, -27.757, 110.684, -15.665, -82.325, 51.133]
  Set speed (1000.0 mm/s)
  MoveL 7485 to (507.65, 494.79, 15.2) mm, rotated rx 0 ry 90 rz 0 deg; joints [-11.389, -27.768, 110.748, -15.426, -82.368, 51.091]
  Set speed (1000.0 mm/s)
  MoveL 7486 to (509.32, 490.68, 15.2) mm, rotated rx 0 ry 90 rz 0 deg; joints [-10.985, -27.75, 110.644, -15.022, -82.272, 51.066]
  Set speed (30.0 mm/s)
  Call Extruder(0.767)
  MoveL 7487 to (490.68, 509.32, 15.2) mm, rotated rx 0 ry 90 rz 0 deg; joints [-13.056, -28.025, 112.396, -17.057, -83.755, 50.877]
  MoveL 7488 to (490.56, 509.44, 15.2) mm, rotated rx 0 ry 90 rz 0 deg; joints [-13.07, -28.026, 112.407, -17.071, -83.764, 50.875]
  Set speed (120.0 mm/s)
  MoveL 7489 to (504.06, 492.37, 15.2) mm, rotated rx 0 ry 90 rz 0 deg; joints [-11.234, -27.847, 111.238, -15.255, -82.759, 50.964]
  Set speed (1000.0 mm/s)
  MoveL 7490 to (503.99, 492.3, 15.2) mm, rotated rx 0 ry 90 rz 0 deg; joints [-11.229, -27.849, 111.248, -15.25, -82.767, 50.961]
  Set speed (15.0 mm/s)
  Call Extruder(0.010)
  MoveL 7491 to (503.99, 491.95, 15.2) mm, rotated rx 0 ry 90 rz 0 deg; joints [-11.197, -27.85, 111.256, -15.218, -82.773, 50.955]
  Call Extruder(0.035)
  MoveL 7492 to (503.98, 490.75, 15.2) mm, rotated rx 0 ry 90 rz 0 deg; joints [-11.087, -27.854, 111.285, -15.106, -82.793, 50.937]
  Call Extruder(0.010)
  MoveL 7493 to (503.98, 490.4, 15.2) mm, rotated rx 0 ry 90 rz 0 deg; joints [-11.054, -27.856, 111.293, -15.073, -82.799, 50.931]
  Call Extruder(0.007)
  MoveL 7494 to (504.33, 490.4, 15.2) mm, rotated rx 0 ry 90 rz 0 deg; joints [-11.048, -27.849, 111.251, -15.068, -82.764, 50.94]
  Call Extruder(0.153)
  MoveL 7495 to (509.6, 490.4, 15.2) mm, rotated rx 0 ry 90 rz 0 deg; joints [-10.955, -27.746, 110.617, -14.992, -82.249, 51.068]
  Call Extruder(0.129)
  MoveL 7496 to (509.6, 494.82, 15.2) mm, rotated rx 0 ry 90 rz 0 deg; joints [-11.356, -27.728, 110.512, -15.4, -82.177, 51.14]
  Call Extruder(0.046)
  MoveL 7497 to (508.02, 494.82, 15.2) mm, rotated rx 0 ry 90 rz 0 deg; joints [-11.385, -27.76, 110.702, -15.423, -82.331, 51.101]
  Call Extruder(0.010)
  MoveL 7498 to (507.67, 494.82, 15.2) mm, rotated rx 0 ry 90 rz 0 deg; joints [-11.391, -27.767, 110.744, -15.428, -82.365, 51.092]
  Call Extruder(0.007)
  MoveL 7499 to (507.67, 495.17, 15.2) mm, rotated rx 0 ry 90 rz 0 deg; joints [-11.423, -27.765, 110.735, -15.461, -82.359, 51.098]
  Call Extruder(0.063)
  MoveL 7500 to (507.68, 497.35, 15.2) mm, rotated rx 0 ry 90 rz 0 deg; joints [-11.621, -27.757, 110.682, -15.662, -82.323, 51.134]
  Call Extruder(0.056)
  MoveL 7501 to (509.6, 497.35, 15.2) mm, rotated rx 0 ry 90 rz 0 deg; joints [-11.585, -27.718, 110.45, -15.633, -82.135, 51.182]
  Call Extruder(0.116)
  MoveL 7502 to (509.6, 501.34, 15.2) mm, rotated rx 0 ry 90 rz 0 deg; joints [-11.946, -27.701, 110.349, -16, -82.067, 51.25]
  Call Extruder(0.010)
  MoveL 7503 to (509.6, 501.69, 15.2) mm, rotated rx 0 ry 90 rz 0 deg; joints [-11.977, -27.7, 110.34, -16.032, -82.061, 51.256]
  Call Extruder(0.007)
  MoveL 7504 to (509.25, 501.69, 15.2) mm, rotated rx 0 ry 90 rz 0 deg; joints [-11.984, -27.707, 110.383, -16.037, -82.095, 51.247]
  Call Extruder(0.036)
  MoveL 7505 to (508.02, 501.69, 15.2) mm, rotated rx 0 ry 90 rz 0 deg; joints [-12.007, -27.732, 110.531, -16.056, -82.215, 51.215]
  Call Extruder(0.010)
  MoveL 7506 to (507.67, 501.69, 15.2) mm, rotated rx 0 ry 90 rz 0 deg; joints [-12.014, -27.739, 110.573, -16.062, -82.249, 51.206]
  Call Extruder(0.007)
  MoveL 7507 to (507.67, 502.04, 15.2) mm, rotated rx 0 ry 90 rz 0 deg; joints [-12.046, -27.737, 110.564, -16.094, -82.243, 51.212]
  Call Extruder(0.063)
  MoveL 7508 to (507.67, 504.2, 15.2) mm, rotated rx 0 ry 90 rz 0 deg; joints [-12.241, -27.728, 110.508, -16.293, -82.205, 51.249]
  Call Extruder(0.056)
  MoveL 7509 to (509.6, 504.21, 15.2) mm, rotated rx 0 ry 90 rz 0 deg; joints [-12.203, -27.689, 110.275, -16.262, -82.018, 51.299]
  Call Extruder(0.157)
  MoveL 7510 to (509.6, 509.6, 15.2) mm, rotated rx 0 ry 90 rz 0 deg; joints [-12.688, -27.664, 110.132, -16.756, -81.922, 51.394]
  Call Extruder(0.559)
  MoveL 7511 to (490.4, 509.6, 15.2) mm, rotated rx 0 ry 90 rz 0 deg; joints [-13.088, -28.028, 112.421, -17.089, -83.776, 50.873]
  MoveL 7512 to (490.4, 490.4, 15.2) mm, rotated rx 0 ry 90 rz 0 deg; joints [-11.303, -28.099, 112.912, -15.282, -84.133, 50.594]
  Call Extruder(0.133)
  MoveL 7513 to (494.98, 490.4, 15.2) mm, rotated rx 0 ry 90 rz 0 deg; joints [-11.218, -28.021, 112.369, -15.21, -83.683, 50.709]
  Call Extruder(0.010)
  MoveL 7514 to (495.33, 490.4, 15.2) mm, rotated rx 0 ry 90 rz 0 deg; joints [-11.212, -28.015, 112.327, -15.204, -83.648, 50.717]
  Call Extruder(0.007)
  MoveL 7515 to (495.33, 490.75, 15.2) mm, rotated rx 0 ry 90 rz 0 deg; joints [-11.244, -28.013, 112.319, -15.237, -83.642, 50.722]
  Call Extruder(0.035)
  MoveL 7516 to (495.33, 491.95, 15.2) mm, rotated rx 0 ry 90 rz 0 deg; joints [-11.356, -28.009, 112.291, -15.35, -83.622, 50.74]
  Call Extruder(0.010)
  MoveL 7517 to (495.32, 492.3, 15.2) mm, rotated rx 0 ry 90 rz 0 deg; joints [-11.388, -28.008, 112.282, -15.383, -83.616, 50.745]
  Call Extruder(0.007)
  MoveL 7518 to (495.68, 492.3, 15.2) mm, rotated rx 0 ry 90 rz 0 deg; joints [-11.382, -28.002, 112.241, -15.378, -83.582, 50.754]
  Call Extruder(0.061)
  MoveL 7519 to (497.78, 492.3, 15.2) mm, rotated rx 0 ry 90 rz 0 deg; joints [-11.343, -27.964, 111.99, -15.345, -83.375, 50.806]
  Call Extruder(0.055)
  MoveL 7520 to (497.78, 490.4, 15.2) mm, rotated rx 0 ry 90 rz 0 deg; joints [-11.167, -27.971, 112.035, -15.167, -83.407, 50.779]
  Call Extruder(0.109)
  MoveL 7521 to (501.54, 490.4, 15.2) mm, rotated rx 0 ry 90 rz 0 deg; joints [-11.098, -27.902, 111.585, -15.11, -83.038, 50.872]
  Call Extruder(0.034)
  MoveL 7522 to (501.54, 491.56, 15.2) mm, rotated rx 0 ry 90 rz 0 deg; joints [-11.205, -27.898, 111.558, -15.218, -83.019, 50.889]
  Call Extruder(0.022)
  MoveL 7523 to (501.54, 492.3, 15.2) mm, rotated rx 0 ry 90 rz 0 deg; joints [-11.273, -27.895, 111.54, -15.287, -83.006, 50.9]
  Call Extruder(0.061)
  MoveL 7524 to (503.64, 492.3, 15.2) mm, rotated rx 0 ry 90 rz 0 deg; joints [-11.235, -27.855, 111.29, -15.255, -82.802, 50.952]
  Call Extruder(0.007)
  MoveL 7525 to (503.99, 492.3, 15.2) mm, rotated rx 0 ry 90 rz 0 deg; joints [-11.229, -27.849, 111.248, -15.25, -82.767, 50.961]
  Set speed (120.0 mm/s)
  MoveL 7526 to (503.99, 491.95, 15.2) mm, rotated rx 0 ry 90 rz 0 deg; joints [-11.197, -27.85, 111.256, -15.218, -82.773, 50.955]
  Set speed (1000.0 mm/s)
  MoveL 7527 to (503.99, 491.9, 15.2) mm, rotated rx 0 ry 90 rz 0 deg; joints [-11.192, -27.85, 111.257, -15.213, -82.774, 50.955]
  Set speed (1000.0 mm/s)
  MoveL 7528 to (504.69, 491.9, 15.2) mm, rotated rx 0 ry 90 rz 0 deg; joints [-11.179, -27.837, 111.173, -15.202, -82.705, 50.972]
  Set speed (1000.0 mm/s)
  MoveL 7529 to (495.3, 492.33, 15.2) mm, rotated rx 0 ry 90 rz 0 deg; joints [-11.391, -28.008, 112.285, -15.386, -83.618, 50.744]
  Set speed (1000.0 mm/s)
  MoveL 7530 to (490.68, 490.68, 15.2) mm, rotated rx 0 ry 90 rz 0 deg; joints [-11.324, -28.094, 112.872, -15.304, -84.1, 50.605]
  Set speed (1000.0 mm/s)
  MoveL 7531 to (490.68, 490.68, 15.3) mm, rotated rx 0 ry 90 rz 0 deg; joints [-11.324, -28.104, 112.877, -15.304, -84.095, 50.606]
  Set speed (30.0 mm/s)
  Call Extruder(0.767)
  MoveL 7532 to (509.32, 509.32, 15.3) mm, rotated rx 0 ry 90 rz 0 deg; joints [-12.669, -27.682, 110.178, -16.735, -81.949, 51.383]
  MoveL 7533 to (509.44, 509.44, 15.3) mm, rotated rx 0 ry 90 rz 0 deg; joints [-12.677, -27.679, 110.16, -16.745, -81.934, 51.389]
  Set speed (120.0 mm/s)
  MoveL 7534 to (507.64, 504.29, 15.3) mm, rotated rx 0 ry 90 rz 0 deg; joints [-12.249, -27.738, 110.514, -16.301, -82.201, 51.251]
  Set speed (1000.0 mm/s)
  MoveL 7535 to (507.39, 502.51, 15.3) mm, rotated rx 0 ry 90 rz 0 deg; joints [-12.093, -27.751, 110.591, -16.142, -82.257, 51.214]
  Set speed (30.0 mm/s)
  Call Extruder(0.280)
  MoveL 7536 to (500.58, 509.32, 15.3) mm, rotated rx 0 ry 90 rz 0 deg; joints [-12.847, -27.855, 111.226, -16.882, -82.792, 51.149]
  Set speed (120.0 mm/s)
  MoveL 7537 to (499.42, 509.32, 15.3) mm, rotated rx 0 ry 90 rz 0 deg; joints [-12.872, -27.877, 111.365, -16.902, -82.904, 51.118]
  Set speed (30.0 mm/s)
  Call Extruder(0.360)
  MoveL 7538 to (490.68, 500.58, 15.3) mm, rotated rx 0 ry 90 rz 0 deg; joints [-12.247, -28.069, 112.633, -16.238, -83.917, 50.746]
  Set speed (120.0 mm/s)
  MoveL 7539 to (490.68, 499.42, 15.3) mm, rotated rx 0 ry 90 rz 0 deg; joints [-12.139, -28.073, 112.662, -16.129, -83.938, 50.729]
  Set speed (30.0 mm/s)
  Call Extruder(0.281)
  MoveL 7540 to (497.52, 492.58, 15.3) mm, rotated rx 0 ry 90 rz 0 deg; joints [-11.373, -27.978, 112.02, -15.375, -83.391, 50.805]
  Set speed (120.0 mm/s)
  MoveL 7541 to (498, 492.1, 15.3) mm, rotated rx 0 ry 90 rz 0 deg; joints [-11.32, -27.971, 111.974, -15.322, -83.352, 50.81]
  Set speed (30.0 mm/s)
  Call Extruder(0.058)
  MoveL 7542 to (499.42, 490.68, 15.3) mm, rotated rx 0 ry 90 rz 0 deg; joints [-11.163, -27.951, 111.838, -15.168, -83.236, 50.825]
  Set speed (120.0 mm/s)
  MoveL 7543 to (500.58, 490.68, 15.3) mm, rotated rx 0 ry 90 rz 0 deg; joints [-11.141, -27.929, 111.699, -15.15, -83.123, 50.853]
  Set speed (30.0 mm/s)
  Call Extruder(0.031)
  MoveL 7544 to (501.33, 491.43, 15.3) mm, rotated rx 0 ry 90 rz 0 deg; joints [-11.197, -27.913, 111.592, -15.209, -83.037, 50.883]
  Set speed (120.0 mm/s)
  MoveL 7545 to (502.48, 492.58, 15.3) mm, rotated rx 0 ry 90 rz 0 deg; joints [-11.282, -27.887, 111.427, -15.299, -82.905, 50.929]
  Set speed (30.0 mm/s)
  Call Extruder(0.202)
  MoveL 7546 to (507.4, 497.5, 15.3) mm, rotated rx 0 ry 90 rz 0 deg; joints [-11.639, -27.772, 110.717, -15.68, -82.342, 51.131]
  Set speed (120.0 mm/s)
  MoveL 7547 to (507.47, 497.57, 15.3) mm, rotated rx 0 ry 90 rz 0 deg; joints [-11.644, -27.77, 110.706, -15.685, -82.334, 51.134]
  Set speed (30.0 mm/s)
  Call Extruder(0.076)
  MoveL 7548 to (509.32, 499.42, 15.3) mm, rotated rx 0 ry 90 rz 0 deg; joints [-11.777, -27.725, 110.437, -15.828, -82.123, 51.211]
  Set speed (120.0 mm/s)
  MoveL 7549 to (509.32, 500.58, 15.3) mm, rotated rx 0 ry 90 rz 0 deg; joints [-11.882, -27.721, 110.408, -15.934, -82.103, 51.231]
  Set speed (30.0 mm/s)
  Call Extruder(0.037)
  MoveL 7550 to (508.43, 501.47, 15.3) mm, rotated rx 0 ry 90 rz 0 deg; joints [-11.979, -27.735, 110.492, -16.03, -82.174, 51.223]
  Set speed (120.0 mm/s)
  MoveL 7551 to (507.65, 497.32, 15.3) mm, rotated rx 0 ry 90 rz 0 deg; joints [-11.618, -27.768, 110.691, -15.66, -82.321, 51.134]
  Set speed (1000.0 mm/s)
  MoveL 7552 to (507.65, 494.73, 15.3) mm, rotated rx 0 ry 90 rz 0 deg; joints [-11.384, -27.778, 110.754, -15.421, -82.364, 51.092]
  Set speed (1000.0 mm/s)
  MoveL 7553 to (509.32, 490.68, 15.3) mm, rotated rx 0 ry 90 rz 0 deg; joints [-10.985, -27.761, 110.649, -15.022, -82.267, 51.067]
  Set speed (30.0 mm/s)
  Call Extruder(0.767)
  MoveL 7554 to (490.68, 509.32, 15.3) mm, rotated rx 0 ry 90 rz 0 deg; joints [-13.056, -28.035, 112.401, -17.058, -83.75, 50.878]
  MoveL 7555 to (490.56, 509.44, 15.3) mm, rotated rx 0 ry 90 rz 0 deg; joints [-13.07, -28.037, 112.412, -17.071, -83.759, 50.877]
  Set speed (120.0 mm/s)
  MoveL 7556 to (504.12, 492.37, 15.3) mm, rotated rx 0 ry 90 rz 0 deg; joints [-11.233, -27.856, 111.235, -15.255, -82.748, 50.967]
  Set speed (1000.0 mm/s)
  MoveL 7557 to (504.05, 492.3, 15.3) mm, rotated rx 0 ry 90 rz 0 deg; joints [-11.227, -27.858, 111.245, -15.249, -82.756, 50.964]
  Set speed (15.0 mm/s)
  Call Extruder(0.010)
  MoveL 7558 to (504.05, 491.95, 15.3) mm, rotated rx 0 ry 90 rz 0 deg; joints [-11.195, -27.859, 111.253, -15.217, -82.762, 50.958]
  Call Extruder(0.035)
  MoveL 7559 to (504.05, 490.75, 15.3) mm, rotated rx 0 ry 90 rz 0 deg; joints [-11.085, -27.864, 111.282, -15.105, -82.781, 50.94]
  Call Extruder(0.010)
  MoveL 7560 to (504.05, 490.4, 15.3) mm, rotated rx 0 ry 90 rz 0 deg; joints [-11.053, -27.865, 111.29, -15.073, -82.787, 50.934]
  Call Extruder(0.007)
  MoveL 7561 to (504.4, 490.4, 15.3) mm, rotated rx 0 ry 90 rz 0 deg; joints [-11.047, -27.858, 111.248, -15.068, -82.753, 50.943]
  Call Extruder(0.151)
  MoveL 7562 to (509.6, 490.4, 15.3) mm, rotated rx 0 ry 90 rz 0 deg; joints [-10.955, -27.756, 110.622, -14.992, -82.244, 51.069]
  Call Extruder(0.127)
  MoveL 7563 to (509.6, 494.76, 15.3) mm, rotated rx 0 ry 90 rz 0 deg; joints [-11.35, -27.739, 110.518, -15.394, -82.173, 51.14]
  Call Extruder(0.056)
  MoveL 7564 to (507.67, 494.76, 15.3) mm, rotated rx 0 ry 90 rz 0 deg; joints [-11.386, -27.778, 110.75, -15.423, -82.361, 51.093]
  Call Extruder(0.074)
  MoveL 7565 to (507.68, 497.29, 15.3) mm, rotated rx 0 ry 90 rz 0 deg; joints [-11.615, -27.767, 110.688, -15.657, -82.318, 51.134]
  Call Extruder(0.056)
  MoveL 7566 to (509.6, 497.29, 15.3) mm, rotated rx 0 ry 90 rz 0 deg; joints [-11.58, -27.729, 110.456, -15.628, -82.131, 51.182]
  Call Extruder(0.120)
  MoveL 7567 to (509.6, 501.4, 15.3) mm, rotated rx 0 ry 90 rz 0 deg; joints [-11.951, -27.711, 110.353, -16.005, -82.061, 51.252]
  Call Extruder(0.010)
  MoveL 7568 to (509.6, 501.75, 15.3) mm, rotated rx 0 ry 90 rz 0 deg; joints [-11.982, -27.71, 110.344, -16.037, -82.055, 51.258]
  Call Extruder(0.007)
  MoveL 7569 to (509.25, 501.75, 15.3) mm, rotated rx 0 ry 90 rz 0 deg; joints [-11.989, -27.717, 110.386, -16.043, -82.089, 51.249]
  Call Extruder(0.036)
  MoveL 7570 to (508.02, 501.75, 15.3) mm, rotated rx 0 ry 90 rz 0 deg; joints [-12.012, -27.742, 110.534, -16.061, -82.209, 51.217]
  Call Extruder(0.010)
  MoveL 7571 to (507.67, 501.75, 15.3) mm, rotated rx 0 ry 90 rz 0 deg; joints [-12.019, -27.749, 110.576, -16.067, -82.243, 51.208]
  Call Extruder(0.007)
  MoveL 7572 to (507.67, 502.1, 15.3) mm, rotated rx 0 ry 90 rz 0 deg; joints [-12.051, -27.747, 110.567, -16.099, -82.236, 51.214]
  Call Extruder(0.063)
  MoveL 7573 to (507.67, 504.26, 15.3) mm, rotated rx 0 ry 90 rz 0 deg; joints [-12.246, -27.738, 110.512, -16.298, -82.199, 51.251]
  Call Extruder(0.056)
  MoveL 7574 to (509.6, 504.26, 15.3) mm, rotated rx 0 ry 90 rz 0 deg; joints [-12.209, -27.699, 110.279, -16.268, -82.012, 51.301]
  Call Extruder(0.155)
  MoveL 7575 to (509.6, 509.6, 15.3) mm, rotated rx 0 ry 90 rz 0 deg; joints [-12.688, -27.675, 110.137, -16.757, -81.916, 51.396]
  Call Extruder(0.559)
  MoveL 7576 to (490.4, 509.6, 15.3) mm, rotated rx 0 ry 90 rz 0 deg; joints [-13.088, -28.039, 112.426, -17.089, -83.771, 50.875]
  MoveL 7577 to (490.4, 490.4, 15.3) mm, rotated rx 0 ry 90 rz 0 deg; joints [-11.303, -28.11, 112.917, -15.282, -84.127, 50.595]
  Call Extruder(0.132)
  MoveL 7578 to (494.92, 490.4, 15.3) mm, rotated rx 0 ry 90 rz 0 deg; joints [-11.219, -28.032, 112.381, -15.211, -83.683, 50.709]
  Call Extruder(0.010)
  MoveL 7579 to (495.27, 490.4, 15.3) mm, rotated rx 0 ry 90 rz 0 deg; joints [-11.213, -28.026, 112.339, -15.205, -83.648, 50.718]
  Call Extruder(0.007)
  MoveL 7580 to (495.27, 490.75, 15.3) mm, rotated rx 0 ry 90 rz 0 deg; joints [-11.245, -28.025, 112.331, -15.238, -83.642, 50.723]
  Call Extruder(0.035)
  MoveL 7581 to (495.27, 491.95, 15.3) mm, rotated rx 0 ry 90 rz 0 deg; joints [-11.357, -28.021, 112.302, -15.351, -83.622, 50.74]
  Call Extruder(0.010)
  MoveL 7582 to (495.27, 492.3, 15.3) mm, rotated rx 0 ry 90 rz 0 deg; joints [-11.389, -28.02, 112.294, -15.384, -83.616, 50.745]
  Call Extruder(0.007)
  MoveL 7583 to (495.62, 492.3, 15.3) mm, rotated rx 0 ry 90 rz 0 deg; joints [-11.383, -28.013, 112.252, -15.379, -83.582, 50.754]
  Call Extruder(0.061)
  MoveL 7584 to (497.72, 492.3, 15.3) mm, rotated rx 0 ry 90 rz 0 deg; joints [-11.344, -27.976, 112.002, -15.346, -83.375, 50.806]
  Call Extruder(0.055)
  MoveL 7585 to (497.72, 490.4, 15.3) mm, rotated rx 0 ry 90 rz 0 deg; joints [-11.168, -27.982, 112.047, -15.168, -83.407, 50.779]
  Call Extruder(0.113)
  MoveL 7586 to (501.61, 490.4, 15.3) mm, rotated rx 0 ry 90 rz 0 deg; joints [-11.097, -27.911, 111.583, -15.109, -83.027, 50.875]
  Call Extruder(0.035)
  MoveL 7587 to (501.61, 491.6, 15.3) mm, rotated rx 0 ry 90 rz 0 deg; joints [-11.208, -27.907, 111.555, -15.221, -83.007, 50.893]
  Call Extruder(0.020)
  MoveL 7588 to (501.61, 492.3, 15.3) mm, rotated rx 0 ry 90 rz 0 deg; joints [-11.272, -27.904, 111.538, -15.286, -82.995, 50.903]
  Call Extruder(0.061)
  MoveL 7589 to (503.7, 492.3, 15.3) mm, rotated rx 0 ry 90 rz 0 deg; joints [-11.234, -27.865, 111.287, -15.254, -82.79, 50.955]
  Call Extruder(0.007)
  MoveL 7590 to (504.05, 492.3, 15.3) mm, rotated rx 0 ry 90 rz 0 deg; joints [-11.227, -27.858, 111.245, -15.249, -82.756, 50.964]
  Set speed (120.0 mm/s)
  MoveL 7591 to (504.05, 491.95, 15.3) mm, rotated rx 0 ry 90 rz 0 deg; joints [-11.195, -27.859, 111.253, -15.217, -82.762, 50.958]
  Set speed (1000.0 mm/s)
  MoveL 7592 to (504.05, 491.9, 15.3) mm, rotated rx 0 ry 90 rz 0 deg; joints [-11.191, -27.859, 111.255, -15.212, -82.762, 50.958]
  Set speed (1000.0 mm/s)
  MoveL 7593 to (504.75, 491.9, 15.3) mm, rotated rx 0 ry 90 rz 0 deg; joints [-11.178, -27.846, 111.171, -15.202, -82.694, 50.975]
  Set speed (1000.0 mm/s)
  MoveL 7594 to (495.24, 492.33, 15.3) mm, rotated rx 0 ry 90 rz 0 deg; joints [-11.392, -28.02, 112.297, -15.387, -83.618, 50.744]
  Set speed (1000.0 mm/s)
  MoveL 7595 to (490.68, 490.68, 15.3) mm, rotated rx 0 ry 90 rz 0 deg; joints [-11.324, -28.104, 112.877, -15.304, -84.095, 50.606]
  Set speed (1000.0 mm/s)
  MoveL 7596 to (490.68, 490.68, 15.4) mm, rotated rx 0 ry 90 rz 0 deg; joints [-11.324, -28.115, 112.882, -15.304, -84.09, 50.608]
  Set speed (30.0 mm/s)
  Call Extruder(0.767)
  MoveL 7597 to (509.32, 509.32, 15.4) mm, rotated rx 0 ry 90 rz 0 deg; joints [-12.669, -27.692, 110.184, -16.736, -81.943, 51.385]
  MoveL 7598 to (509.44, 509.44, 15.4) mm, rotated rx 0 ry 90 rz 0 deg; joints [-12.677, -27.689, 110.165, -16.745, -81.929, 51.39]
  Set speed (120.0 mm/s)
  MoveL 7599 to (507.64, 504.34, 15.4) mm, rotated rx 0 ry 90 rz 0 deg; joints [-12.254, -27.749, 110.518, -16.307, -82.195, 51.254]
  Set speed (1000.0 mm/s)
  MoveL 7600 to (507.39, 502.51, 15.4) mm, rotated rx 0 ry 90 rz 0 deg; joints [-12.093, -27.762, 110.596, -16.142, -82.251, 51.216]
  Set speed (30.0 mm/s)
  Call Extruder(0.280)
  MoveL 7601 to (500.58, 509.32, 15.4) mm, rotated rx 0 ry 90 rz 0 deg; joints [-12.847, -27.865, 111.231, -16.882, -82.787, 51.151]
  Set speed (120.0 mm/s)
  MoveL 7602 to (499.42, 509.32, 15.4) mm, rotated rx 0 ry 90 rz 0 deg; joints [-12.872, -27.887, 111.37, -16.902, -82.899, 51.119]
  Set speed (30.0 mm/s)
  Call Extruder(0.360)
  MoveL 7603 to (490.68, 500.58, 15.4) mm, rotated rx 0 ry 90 rz 0 deg; joints [-12.247, -28.08, 112.638, -16.238, -83.912, 50.748]
  Set speed (120.0 mm/s)
  MoveL 7604 to (490.68, 499.42, 15.4) mm, rotated rx 0 ry 90 rz 0 deg; joints [-12.139, -28.084, 112.668, -16.129, -83.933, 50.731]
  Set speed (30.0 mm/s)
  Call Extruder(0.281)
  MoveL 7605 to (497.52, 492.58, 15.4) mm, rotated rx 0 ry 90 rz 0 deg; joints [-11.373, -27.989, 112.025, -15.376, -83.386, 50.807]
  Set speed (120.0 mm/s)
  MoveL 7606 to (497.94, 492.15, 15.4) mm, rotated rx 0 ry 90 rz 0 deg; joints [-11.326, -27.983, 111.984, -15.329, -83.351, 50.811]
  Set speed (30.0 mm/s)
  Call Extruder(0.061)
  MoveL 7607 to (499.42, 490.68, 15.4) mm, rotated rx 0 ry 90 rz 0 deg; joints [-11.163, -27.961, 111.843, -15.168, -83.231, 50.826]
  Set speed (120.0 mm/s)
  MoveL 7608 to (500.58, 490.68, 15.4) mm, rotated rx 0 ry 90 rz 0 deg; joints [-11.141, -27.94, 111.704, -15.151, -83.117, 50.855]
  Set speed (30.0 mm/s)
  Call Extruder(0.033)
  MoveL 7609 to (501.39, 491.49, 15.4) mm, rotated rx 0 ry 90 rz 0 deg; joints [-11.201, -27.922, 111.588, -15.214, -83.024, 50.887]
  Set speed (120.0 mm/s)
  MoveL 7610 to (502.48, 492.58, 15.4) mm, rotated rx 0 ry 90 rz 0 deg; joints [-11.282, -27.897, 111.432, -15.299, -82.899, 50.931]
  Set speed (30.0 mm/s)
  Call Extruder(0.202)
  MoveL 7611 to (507.4, 497.5, 15.4) mm, rotated rx 0 ry 90 rz 0 deg; joints [-11.639, -27.783, 110.722, -15.68, -82.337, 51.132]
  Set speed (120.0 mm/s)
  MoveL 7612 to (507.41, 497.51, 15.4) mm, rotated rx 0 ry 90 rz 0 deg; joints [-11.64, -27.782, 110.719, -15.681, -82.335, 51.133]
  Set speed (30.0 mm/s)
  Call Extruder(0.078)
  MoveL 7613 to (509.32, 499.42, 15.4) mm, rotated rx 0 ry 90 rz 0 deg; joints [-11.777, -27.736, 110.442, -15.828, -82.117, 51.213]
  Set speed (120.0 mm/s)
  MoveL 7614 to (509.32, 500.58, 15.4) mm, rotated rx 0 ry 90 rz 0 deg; joints [-11.882, -27.731, 110.413, -15.934, -82.098, 51.232]
  Set speed (30.0 mm/s)
  Call Extruder(0.039)
  MoveL 7615 to (508.37, 501.52, 15.4) mm, rotated rx 0 ry 90 rz 0 deg; joints [-11.985, -27.746, 110.503, -16.036, -82.173, 51.224]
  Set speed (120.0 mm/s)
  MoveL 7616 to (507.65, 497.26, 15.4) mm, rotated rx 0 ry 90 rz 0 deg; joints [-11.613, -27.778, 110.697, -15.654, -82.316, 51.134]
  Set speed (1000.0 mm/s)
  MoveL 7617 to (507.65, 494.67, 15.4) mm, rotated rx 0 ry 90 rz 0 deg; joints [-11.378, -27.789, 110.761, -15.416, -82.36, 51.092]
  Set speed (1000.0 mm/s)
  MoveL 7618 to (509.32, 490.68, 15.4) mm, rotated rx 0 ry 90 rz 0 deg; joints [-10.985, -27.771, 110.654, -15.022, -82.261, 51.068]
  Set speed (30.0 mm/s)
  Call Extruder(0.767)
  MoveL 7619 to (490.68, 509.32, 15.4) mm, rotated rx 0 ry 90 rz 0 deg; joints [-13.056, -28.046, 112.406, -17.058, -83.744, 50.88]
  MoveL 7620 to (490.56, 509.44, 15.4) mm, rotated rx 0 ry 90 rz 0 deg; joints [-13.07, -28.048, 112.417, -17.071, -83.754, 50.879]
